# B&R Automation Studio project TD52 (part 122)

### module_HC.typ - Package data types
```iecst
TYPE
	IN_HC_Struct : 	STRUCT
		tAB2HC : AmmBase2MM;
		tPB2MM : ParaBase2MM_type;
		tCtr_Cust1_Out : _tGeACtrOut; (*controller customized*) (*OldName:REG1; Cycle:5;*)
		tCtr_Cust2_Out : _tGeACtrOut; (*controller customized*) (*OldName:REG2; Cycle:5;*)
		tCtr_Cust3_Out : _tGeACtrOut; (*controller customized*) (*OldName:REG3; Cycle:5;*)
		tCtr_Cust4_Out : _tGeACtrOut; (*controller customized*) (*OldName:REG4; Cycle:5;*)
		tCtr_Cust5_Out : _tGeACtrOut; (*controller customized*) (*OldName:REG5; Cycle:5;*)
		tCtr_Cust6_Out : _tGeACtrOut; (*controller customized*) (*OldName:REG6; Cycle:5;*)
		tCtr_Cust7_Out : _tGeACtrOut; (*controller customized*) (*OldName:REG7; Cycle:5;*)
		tCtr_Cust8_Out : _tGeACtrOut; (*controller customized*) (*OldName:REG8; Cycle:5;*)
		tCtr_Cust1_In : _tGeACtrIn; (*controller customized*) (*OldName:F_SPSR1; Cycle:5;*)
		tCtr_Cust2_In : _tGeACtrIn; (*controller customized*) (*OldName:F_SPSR2; Cycle:5;*)
		tCtr_Cust3_In : _tGeACtrIn; (*controller customized*) (*OldName:F_SPSR3; Cycle:5;*)
		tCtr_Cust4_In : _tGeACtrIn; (*controller customized*) (*OldName:F_SPSR4; Cycle:5;*)
		tCtr_Cust5_In : _tGeACtrIn; (*controller customized*) (*OldName:F_SPSR5; Cycle:5;*)
		tCtr_Cust6_In : _tGeACtrIn; (*controller customized*) (*OldName:F_SPSR6; Cycle:5;*)
		tCtr_Cust7_In : _tGeACtrIn; (*controller customized*) (*OldName:F_SPSR7; Cycle:5;*)
		tCtr_Cust8_In : _tGeACtrIn; (*controller customized*) (*OldName:F_SPSR8; Cycle:5;*)
		rCust_SparePara : ARRAY[0..200]OF REAL; (*SPS_REZP1 to SPS_REZP200	*) (* OldName: SPS_REZP1, SPS_REZP2, SPS_REZP70; Cycle: 5; *)
		tCustAnaIn : ARRAY[0..120]OF HALioAi_Type; (*Replacement for RAN_KANAL...*) (*OldName: ANA_RAN	; Cycle: 5;*)
		tCustDigIn : ARRAY[0..200]OF HALioDi_Type; (*new, reserved for Project specific use*) (*OldName: new PV	; Cycle: 5;*)
		tT_ECW_Ext_Hi : HALioDi_Type; (*DI temperature engine cooling water high external*) (*OldName:KTMA; Cycle:5;*)
		tEC_Failure : HALioDi_Type; (*DI emergency cooler failure*) (*OldName:ST_K; Cycle:5;*)
		tChC_Failure : HALioDi_Type; (*DI charge cooler failure*) (*OldName:ST_GKV; Cycle:5;*)
		tPr_CCircuit_Lo : HALioDi_Type; (*DI water pressure cooler circuit low*) (*OldName:WDK; Cycle:5;*)
		tPr_HW_Lo : HALioDi_Type; (*DI heat water pressure low*) (*OldName:HWD; Cycle:5;*)
		tPr_ChC_Lo : HALioDi_Type; (*DI charge cooler water pressure low*) (*OldName:GKWD; Cycle:5;*)
		tGCB_On : HALioDi_Type; (*DI generator circuit breaker closed*) (*OldName:GCB_ON; Cycle:5;*)
		tT_AirOutdoor : HALioAi_Type; (*AI temperature air outdoor*) (*OldName:ANA_ULT; Cycle:5;*)
		tPr_ECW : HALioAi_Type; (*pressure engine cooling water M.04-PI-001*) (*OldName:ANA.KWD; Cycle:5;*)
		tPr_ECWaEng : HALioAi_Type; (*pressure engine cooling water after engine M.04-PI-058*) (*OldName:AI_p_ECWaEng; Cycle:5;*)
		tT_ECW : HALioAi_Type; (*temperature engine cooling water M.04-TI-001*) (*OldName:ANA.KWT; Cycle:5;*)
		tT_HW_ReBeEng : HALioAi_Type; (*temperature heat water return before engine M.06-TI-001*) (*OldName:ANA.RLT_M; Cycle:5;*)
		tT_HW_ReAfEC : HALioAi_Type; (*temperature heat water return after emergency cooler P.06-TI-015, M.04-TI-015*) (*OldName:ANA.RLT_NK; Cycle:5;*)
		tT_HW_Re : HALioAi_Type; (*temperature heat water return P.06-TI-012, M.04-TI-012*) (*OldName:ANA.RLTP; Cycle:5;*)
		tT_HW_Su : HALioAi_Type; (*temperature heat water supply P.06-TI-014, M.04-TI-014*) (*OldName:ANA.VLTP; Cycle:5;*)
		tT_Su_PriCirc : HALioAi_Type; (*AI supply water temperature primary circuit [°C]*) (*OldName: new PV	; Cycle: 5;*)
		tT_Re_PriCirc : HALioAi_Type; (*AI return water temperature primary circuit [°C]*) (*OldName: new PV	; Cycle: 5;*)
		tT_Su_SecCirc : HALioAi_Type; (*AI supply water temperature secondary circuit [°C]*) (*OldName: new PV	; Cycle: 5;*)
		tT_Re_SecCirc : HALioAi_Type; (*AI return water temperature secondary circuit [°C]*) (*OldName: new PV	; Cycle: 5;*)
		tP_Heat : HALioAi_Type; (*AI heating power engine heat water circuit [kW]*) (*OldName: new PV	; Cycle: 5;*)
		tP_Heat_Imp : HALioDi_Type; (*DI heating power engine heat water circuit pulse*) (*OldName: new PV	; Cycle: 5;*)
		rT_Ch_T2s_Avg : REAL; (*average charge temperature t2' [°C]*) (*OldName: newPV; Cycle: 5;*)
		tT_EO : HALioAi_Type; (*temperature engine oil M.03-TI-001*) (*OldName:ANA.OTP; Cycle:5;*)
		tECWP1Dem : HALioDo_Type; (*DO engine cooling water pump 1 demand*) (*OldName:A_MKWP1; Cycle:5;*)
		tPr_HW_Hi1 : HALioDi_Type; (*DI heat water pressure high*) (*OldName:HWDX1; Cycle:5;*)
		tPr_HW_Hi : HALioDi_Type; (*DI heat water pressure high*) (*OldName:HWDX; Cycle:5;*)
		tT_HW_Hi1 : HALioDi_Type; (*DI heat water temperature high P.06-TS-023*) (*OldName:HWTP1; Cycle:5;*)
		tT_HW_Hi : HALioDi_Type; (*DI heat water temperature high P.06-TS-001*) (*OldName:HWTP; Cycle:5;*)
		tFlow_HW_Lo : HALioDi_Type; (*DI heat water flow low*) (*OldName:HWDF; Cycle:5;*)
		tT_ChCW_Hi : HALioDi_Type; (*DI charge cooling water temperature high*) (*OldName:GKWT_2; Cycle:5;*)
		tT_HW_Su_LT : HALioAi_Type; (*temperature heat water supply low temp.circuit [°C] M.07-TI-048*) (*OldName:NT_supply_water_temp; Cycle:5;*)
		tT_ECW_AfEng : HALioAi_Type; (*temperature engine cooling water after engine [°C]*) (*OldName:MKW_press_after_engine; Cycle:5;*)
		tEng_Run : HALioDo_Type; (*engine is running*) (*OldName:M_BTRB; Cycle:5;*)
		tT_HW_Re_LT : HALioAi_Type; (*temperature heat water return low temp.circuit [°C] M.07-TI-001*) (*OldName:iT_HWR_LT; Cycle:5;*)
		tAuxV_ModIf_ok : HALioDi_Type; (*DI auxiliary voltage supply ok Module interface*) (*OldName:SPG_HBT; Cycle:5;*)
		tAuxV_Aux_ok : HALioDi_Type; (*DI auxiliary voltage supply ok Auxiliaries panel*) (*OldName:SPG_HBT; Cycle:5;*)
		tAuxV_Supply_Ok : HALioDi_Type; (*DI auxiliary voltage supply ok*) (*OldName:SPG_HBT; Cycle:5;*)
		tChC_FanRdy : HALioDi_Type; (*DI charge cooler fan ready*) (*OldName:RDY_ICF; Cycle:5;*)
		tPr_HW_Su_LT : HALioAi_Type; (*supply water pressure LT circuit M.07-PI-001*) (*OldName:AI_p_VL_NT; Cycle:5;*)
		tPr_HW_Su_HT : HALioAi_Type; (*supply water pressure HT circuit M.06-PI-001*) (*OldName:AI_p_VL_HT; Cycle:5;*)
		tT_ECWbEng : HALioAi_Type; (*engine cooling water temperature before engine measurement active M.04-TI-002*) (*OldName:newPv; Cycle:5;*)
		tPr_HW_Re_LT : HALioAi_Type; (*pressure heat water return low temp.circuit M.07-PI-002*) (*OldName:newPv; Cycle:5;*)
		tPr_HW_Re_HT : HALioAi_Type; (*pressure heat water return high temp.circuit M.06-PI-002*) (*OldName:newPv; Cycle:5;*)
		tPr_HW_Re_PreH_ECW : HALioAi_Type; (*pressure heat water return preheating engine cooling water M.04-PI-005*) (*OldName:newPv; Cycle:5;*)
		tPr_HW_Re_PreH_EO : HALioAi_Type; (*pressure heat water return preheating engine oil M.03-PI-005*) (*OldName:newPv; Cycle:5;*)
		tPr_EO_Mod_Out : HALioAi_Type; (*pressure engine oil module outlet M.03-PI-006*) (*OldName:newPv; Cycle:5;*)
		tT_ECW_Mod_In : HALioAi_Type; (*temperature engine cooling water, engine cooling water module inlet M.04-TI-003*) (*OldName:newPv; Cycle:5;*)
		tT_ECW_Mod_Out : HALioAi_Type; (*temperature engine cooling water, engine cooling water module outlet M.04-TI-004*) (*OldName:newPv; Cycle:5;*)
		tT_EO_Mod_In : HALioAi_Type; (*temperature engine oil, oil module inlet M.03-TI-004*) (*OldName:newPv; Cycle:5;*)
		tT_EO_Mod_Out : HALioAi_Type; (*temperature engine oil, oil module outlet M.03-TI-003*) (*OldName:newPv; Cycle:5;*)
		tT_HW_Su_PreH_ECW : HALioAi_Type; (*temperature heat water supply preheating engine cooling water M.04-TI-005*) (*OldName:newPv; Cycle:5;*)
		tT_HW_Re_PreH_ECW : HALioAi_Type; (*temperature heat water return preheating engine cooling water M.04-TI-006*) (*OldName:newPv; Cycle:5;*)
		tT_HW_Su_PreH_EO : HALioAi_Type; (*temperature heat water supply preheating engine oil M.03-TI-005*) (*OldName:newPv; Cycle:5;*)
		tT_HW_Re_PreH_EO : HALioAi_Type; (*temperature heat water return preheating engine oil M.03-TI-006*) (*OldName:newPv; Cycle:5;*)
		iSt_OpMode : UDINT; (*engine operating mode*) (*OldName:newPv; Cycle:5;*)
		rN_EngAct : REAL; (*engine speed actual [1/min]*) (*OldName:n_ist; Cycle:5;*)
		rT_ChC_Ctr_Wex : REAL; (*charge temperature controller external setpoint(knocking)*) (*OldName:Wex_GEMREG; Cycle:5;*)
		bEng_Dem_EPS : BOOL; (*engine demand for emergency power supply*) (*OldName:M_NANF; Cycle:5;*)
		bEng_Aux_Dem_CDR : BOOL; (*engine auxiliaries demand with cool down run*) (*OldName:ANFHBT; Cycle:5;*)
		bEng_Aux_Dem : BOOL; (*engine auxiliaries demand*) (*OldName:M_ANFHBT; Cycle:5;*)
		iIdx_OMSS : INT; (*engine operation mode selection*) (*OldName:newPv; Cycle:5;*)
		rP_Act_Norm_Filt : REAL; (*actual power related to rP_Nom filtered(1s) [%] *) (*OldName:P_IST; Cycle:5;*)
		bEC_Rel : BOOL; (*release emergency cooler from monitoring*) (*OldName:K_frg; Cycle:5;*)
		bChC_Rel : BOOL; (*release charge cooler from monitoring*) (*OldName:GK_frg; Cycle:5;*)
		tCDP_Dem : HALioDo_Type; (*demand condensor pump*) (*OldName:newPv; Cycle:5;*)
		tHWF_Fail : HALioDi_Type; (*failure heating circuit flap*) (*OldName:newPv; Cycle:5;*)
		tCDP_Op : HALioDi_Type; (*failure condensor pump*) (*OldName:newPv; Cycle:5;*)
		tT_HW_HC_Re : HALioAi_Type; (*heating circuit return temperature*) (*OldName:newPv; Cycle:5;*)
		tT_CD_Su : HALioAi_Type; (*supply temperature condensor circuit*) (*OldName:newPv; Cycle:5;*)
		tT_CD_Re : HALioAi_Type; (*return temperature condensor circuit*) (*OldName:newPv; Cycle:5;*)
		tPos_HW_ReValve : HALioAi_Type; (*position heating water return temperature regulation valve*) (*OldName:newPv; Cycle:5;*)
		tPos_HW_EC_ReValve : HALioAi_Type; (*position heating water return temperature after cooler regulation valve*) (*OldName:newPv; Cycle:5;*)
		tPos_ChC_Valve : HALioAi_Type; (*position charge temperature regulation valve*) (*OldName:newPv; Cycle:5;*)
		tBHV_Op : HALioDi_Type; (*failure boiler house ventilation*) (*OldName:newPv; Cycle:5;*)
		tDemnd_BHV : HALioDi_Type; (*demand boiler house ventilation*) (*OldName:newPv; Cycle:5;*)
		bMsg1031 : BOOL; (*emergency stop / safety loop*) (*OldName:M_SIS; Cycle:5;*)
		bMsg1053 : BOOL; (*gas alarm*) (*OldName:M_GAL; Cycle:5;*)
		bMsg1054 : BOOL; (*fire alarm*) (*OldName:M_BAL; Cycle:5;*)
		bMsg3003 : BOOL; (*signal failure( 2101 or 2102 or 2103 or 2104 or 3152 > 24h)*) (*OldName:M_MS; Cycle:5;*)
		tManAuxCtr : tManAuxCtr_typ; (*Manual operating auxiliaries control - Handbedienebene*) (*OldName: new PV; Cycle: 5;*)
		tT_ECW_bChC_HT : HALioAi_Type; (*temperature engine cooling water before charge cooler high temp.circ. M.06-TI-014*) (*OldName:newPv; Cycle:5;*)
		tT_ECW_bOilC : HALioAi_Type; (*temperature engine cooling water before oil cooler M.06-TI-020*) (*OldName:newPv; Cycle:5;*)
		tT_ECW_bECWC : HALioAi_Type; (*temperature engine cooling water before engine cooling water cooler M.06-TI-030*) (*OldName:newPv; Cycle:5;*)
		bAMM_T_Ch_T2s_Avg : BOOL; (*collective warning - average charge temp. t2'  *) (*OldName: new PV; Cycle:5;*) (*SWAT920/2*)
		bT_ChC_Ctr_Wex_Enable_Cust : BOOL; (*new V4.5*)
		rT_ChC_Ctr_Wex_Cust : REAL; (*new V4..5*)
		rCustomizedHC : ARRAY[0..99]OF REAL; (*New customizable interface 2017  - BETA PHASE, use only in coordination with TPSS*)
		bChC2_Rel : BOOL; (*release charge cooler 2 from monitoring*) (*OldName:newPV; Cycle:5;*)
		bAMM_T_Ch_T1HP_Avg : BOOL; (*collective warning - average charge temp. before high-pressure TC*) (*OldName: new PV; Cycle:5;*)
		rT_Ch_T1HP_Avg : REAL; (*average charge temperature before high-pressure turbo charger T1-HP [°C]*) (*OldName: newPV; Cycle: 5;*)
		tPos_ChC2_Valve : HALioAi_Type; (*AI Position temperature-regulation-valve 2nd LT charge cooler circuit (T1-HP)*) (*OldName:newPv; Cycle:5;*)
		tPr_ChC2_Lo : HALioDi_Type; (*DI charge cooler 2 water pressure low - DI = FALSE if pressure is low*) (*OldName:newPV; Cycle:5;*)
		tChC2_FanRdy : HALioDi_Type; (*DI charge cooler 2 fan ready*) (*OldName:newPV; Cycle:5;*)
		tChC2_Failure : HALioDi_Type; (*DI charge cooler 2 failure - DI = FALSE if failure active*) (*OldName:newPV; Cycle:5;*)
		tT_ChC2_Su_LT : HALioAi_Type; (*AI supply water temperature 2nd LT charge cooler circuit (T1-HP) [°C] (P.07-TI-004)*) (*OldName:newPV; Cycle:5;*)
		tT_ChC2_Re_LT : HALioAi_Type; (*AI return water temperature 2nd LT charge cooler circuit (T1-HP) [°C] (P.07-TI-006)*) (*OldName:newPV; Cycle:5;*)
		tT_ChC2W_Hi : HALioDi_Type; (*DI charge cooler 2 water temperature high - DI = FALSE if water temp. too high*) (*OldName:newPV; Cycle:5;*)
		tT_HW_EGHE_Hi : HALioDi_Type; (*DI Heating water temperature max. exhaust gas cooler*)
		tT_HW_EGCD_Hi : HALioDi_Type; (*DI Heating water temperature max. exhaust gas condenser*)
		tCust_HW_Ext_Trip : HALioDi_Type; (*DI External heating water circuit monitoring*)
		bECWP_MechDriven : BOOL;  (* CUSTOM for new Pr_ECW plausibility check: Mechanically driven ECWP on type3 or type2 *)
		tECWP_Op : HALioDi_Type; (* DI engine cooling water pump operating *)
		tT_HW_Su_Unit : HALioAi_Type; (*SAFETY PLC: Heating water supply temperature - Unit (M.06-TI-003)*) (*OldName: new PV; Cycle: 5;*) (*V04.25.00.00*)
	END_STRUCT; (*END_IN*)
	OUT_HC_Struct : 	STRUCT
		tChC_Heating : HALioDo_Type; (*DO charge cooler pre heating*) (*OldName:FG_KT; Cycle:5;*)
		tHC2AB : MM2AmmBase;
		tHC2PB : MM2ParaBase_type;
		tExCo_Rel : HALioDo_Type; (*DO external cooler release*) (*OldName:FG_KT; Cycle:5;*)
		tChC_DemPump : HALioDo_Type; (*DO charge cooler demand pump*) (*OldName:GKP_EIN; Cycle:5;*)
		tChC_DemFan1 : HALioDo_Type; (*DO charge cooler demand fan 1*) (*OldName:GKV_1; Cycle:5;*)
		tChC_DemFan2 : HALioDo_Type; (*DO charge cooler demand fan 2*) (*OldName:GKV_2; Cycle:5;*)
		tChC_DemFan3 : HALioDo_Type; (*DO charge cooler demand fan 3*) (*OldName:GKV_3; Cycle:5;*)
		tChC_DemFan4 : HALioDo_Type; (*DO charge cooler demand fan 4*) (*OldName:GKV_4; Cycle:5;*)
		tChC_DemFan5 : HALioDo_Type; (*DO charge cooler demand fan 5*) (*OldName:GKV_5; Cycle:5;*)
		tChC_DemFan6 : HALioDo_Type; (*DO charge cooler demand fan 6*) (*OldName:GKV_6; Cycle:5;*)
		tChC_DemFan7 : HALioDo_Type; (*DO charge cooler demand fan 7*) (*OldName:GKV_7; Cycle:5;*)
		tChC_DemFan8 : HALioDo_Type; (*DO charge cooler demand fan 8*) (*OldName:GKV_8; Cycle:5;*)
		tChC_DemFan9 : HALioDo_Type; (*DO charge cooler demand fan 9*) (*OldName:GKV_9; Cycle:5;*)
		tChC_DemFan10 : HALioDo_Type; (*DO charge cooler demand fan 10*) (*OldName:GKV_10; Cycle:5;*)
		tChC_DemFan11 : HALioDo_Type; (*DO charge cooler demand fan 11*) (*OldName:GKV_11; Cycle:5;*)
		tChC_DemFan12 : HALioDo_Type; (*DO charge cooler demand fan 12*) (*OldName:GKV_12; Cycle:5;*)
		tChC_DemFan13 : HALioDo_Type; (*DO charge cooler demand fan 13*) (*OldName:GKV_13; Cycle:5;*)
		tChC_DemFan14 : HALioDo_Type; (*DO charge cooler demand fan 14*) (*OldName:GKV_14; Cycle:5;*)
		tChC_DemFan15 : HALioDo_Type; (*DO charge cooler demand fan 15*) (*OldName:GKV_15; Cycle:5;*)
		tChC_DemFan16 : HALioDo_Type; (*DO charge cooler demand fan 16*) (*OldName:GKV_16; Cycle:5;*)
		tEC_DemPump : HALioDo_Type; (*DO emergency cooler demand pump*) (*OldName:KP_EIN; Cycle:5;*)
		tEC_DemFan1 : HALioDo_Type; (*DO emergency cooler demand fan 1*) (*OldName:KV_1; Cycle:5;*)
		tEC_DemFan2 : HALioDo_Type; (*DO emergency cooler demand fan 2*) (*OldName:KV_2; Cycle:5;*)
		tEC_DemFan3 : HALioDo_Type; (*DO emergency cooler demand fan 3*) (*OldName:KV_3; Cycle:5;*)
		tEC_DemFan4 : HALioDo_Type; (*DO emergency cooler demand fan 4*) (*OldName:KV_4; Cycle:5;*)
		tEC_DemFan5 : HALioDo_Type; (*DO emergency cooler demand fan 5*) (*OldName:KV_5; Cycle:5;*)
		tEC_DemFan6 : HALioDo_Type; (*DO emergency cooler demand fan 6*) (*OldName:KV_6; Cycle:5;*)
		tEC_DemFan7 : HALioDo_Type; (*DO emergency cooler demand fan 7*) (*OldName:KV_7; Cycle:5;*)
		tEC_DemFan8 : HALioDo_Type; (*DO emergency cooler demand fan 8*) (*OldName:KV_8; Cycle:5;*)
		tEC_DemFan9 : HALioDo_Type; (*DO emergency cooler demand fan 9*) (*OldName:KV_9; Cycle:5;*)
		tEC_DemFan10 : HALioDo_Type; (*DO emergency cooler demand fan 10*) (*OldName:KV_10; Cycle:5;*)
		tEC_DemFan11 : HALioDo_Type; (*DO emergency cooler demand fan 11*) (*OldName:KV_11; Cycle:5;*)
		tEC_DemFan12 : HALioDo_Type; (*DO emergency cooler demand fan 12*) (*OldName:KV_12; Cycle:5;*)
		tEC_DemFan13 : HALioDo_Type; (*DO emergency cooler demand fan 13*) (*OldName:KV_13; Cycle:5;*)
		tEC_DemFan14 : HALioDo_Type; (*DO emergency cooler demand fan 14*) (*OldName:KV_14; Cycle:5;*)
		tEC_DemFan15 : HALioDo_Type; (*DO emergency cooler demand fan 15*) (*OldName:KV_15; Cycle:5;*)
		tEC_DemFan16 : HALioDo_Type; (*DO emergency cooler demand fan 16*) (*OldName:KV_16; Cycle:5;*)
		tECW_DemBpP : HALioDo_Type; (*DO demand engine cooling water bypass pump (AMOT)*) (*OldName:BP_P; Cycle:5;*)
		tECW_DemBpV : HALioDo_Type; (*DO demand engine cooling water bypass valve (AMOT)*) (*OldName:BP_V; Cycle:5;*)
		tCtr_ChC_Set : HALioAo_Type; (*AO charge temperature cooler control valve*) (*OldName:Reg9_y; Cycle:5;*)
		tCtr_HWRe_Set : HALioAo_Type; (*AO heat water return temperature control valve*) (*OldName:Reg10_y; Cycle:5;*)
		tCtr_EC_Set : HALioAo_Type; (*AO heat water return temperature control valve emergency cooler*) (*OldName:Reg11_y; Cycle:5;*)
		tCtr_HWSu_Set : HALioAo_Type; (*AO heat water supply temperature control valve*) (*OldName:Reg14_y; Cycle:5;*)
		tCtr_ChCV_Set : HALioAo_Type; (*AO charge temperature cooler ventilation*) (*OldName:Reg15_y, GKV_y; Cycle:5;*)
		tCtr_ChCHP_Set : HALioAo_Type; (*AO charge temperature cooler high pressure control valve*) (*OldName:Reg18_y; Cycle:5;*)
		bT_ECW_Hi : BOOL; (*temperature engine cooling water limit high*) (*OldName:AN_KTMA; Cycle:5;*)
		bT_ECW_Lo : BOOL; (*temperature engine cooling water limit low*) (*OldName:AN_KTMI; Cycle:5;*)
		bT_ECW_RelLoad : BOOL; (*temperature engine cooling water release load*) (*OldName:AN_LFG; Cycle:5;*)
		bT_ECW_PreH_OFF : BOOL; (*temperature engine cooling water preheating off*) (*OldName:AN_VORW; Cycle:5;*)
		rP_Red_T_HWR_Norm : REAL; (*power reduction heat water return temperature high [% Pnom]*) (*OldName:RED_RLT; Cycle:5;*)
		rP_Red_T_ECW_Norm : REAL; (*power reduction engine cooling water temperature high [% Pnom]*) (*OldName:RED_KWT; Cycle:5;*)
		bPr_ECW_Lo1 : BOOL; (*pressure engine cooling water limit low 1*) (*OldName:AN_KDGW1; Cycle:5;*)
		tHWF_Dem : HALioDo_Type; (*demand heating circuit flap*) (*OldName:newPv; Cycle:5;*)
		tCtr_CDSu_Set : HALioAo_Type; (*setpoint frequency conferter condensor pump*) (*OldName:newPv; Cycle:5;*)
		tBHV_Dem : HALioDo_Type; (*demand boiler house ventilation*) (*OldName:newPv; Cycle:5;*)
		iCnt_P_Heat : DINT; (*counter heating power engine heat water circuit*) (*OldName:newPv; Cycle:5;*)
		bMsg1019 : BOOL; (*engine cooling water pressure low*) (*OldName:M_KDMI; Cycle:5;*)
		bMsg2104 : BOOL; (*signal failure engine cooling water pressure *) (*OldName:M_MSKWD; Cycle:5;*)
		bMsg2101 : BOOL; (*signal failure engine cooling water temperature*) (*OldName:M_MSKWT; Cycle:5;*)
		bMsg3404 : BOOL; (*water pressure cooler circuit low*) (*OldName:M_NKWD_W; Cycle:5;*)
		bMsg1130 : BOOL; (*charge cooler water pressure low*) (*OldName:AMM_A11xx[]; Cycle:5;*)
		bMsg2117 : BOOL; (*charge cooler water pressure low*) (*OldName:M_GKWD; Cycle:5;*)
		rP_Red_T_ECW_Low_Norm : REAL; (*power reduction engine cooling water temperature low [% Pnom]*) (*OldName:newPv; Cycle:5;*)
		rCustomizedHC : ARRAY[0..99]OF REAL; (*New customizable interface 2017  - BETA PHASE, use only in coordination with TPSS*)
		tChC2_DemPump : HALioDo_Type; (*DO charge cooler 2 demand pump*) (*OldName:newPV; Cycle:5;*)
		tCtr_ChC2_Valve_Set : HALioAo_Type; (*AO Control temperature-regulation-valve 2nd LT charge cooler circuit (T1-HP)*) (*OldName:newPV; Cycle:5;*)
		tChC2_DemFan1 : HALioDo_Type; (*DO charge cooler 2 demand fan 1*) (*OldName:newPV; Cycle:5;*)
		tChC2_DemFan2 : HALioDo_Type; (*DO charge cooler 2 demand fan 2*) (*OldName:newPV; Cycle:5;*)
		tChC2_DemFan3 : HALioDo_Type; (*DO charge cooler 2 demand fan 3*) (*OldName:newPV; Cycle:5;*)
		tChC2_DemFan4 : HALioDo_Type; (*DO charge cooler 2 demand fan 4*) (*OldName:newPV; Cycle:5;*)
		tChC2_DemFan5 : HALioDo_Type; (*DO charge cooler 2 demand fan 5*) (*OldName:newPV; Cycle:5;*)
		tChC2_DemFan6 : HALioDo_Type; (*DO charge cooler 2 demand fan 6*) (*OldName:newPV; Cycle:5;*)
		tChC2_DemFan7 : HALioDo_Type; (*DO charge cooler 2 demand fan 7*) (*OldName:newPV; Cycle:5;*)
		tChC2_DemFan8 : HALioDo_Type; (*DO charge cooler 2 demand fan 8*) (*OldName:newPV; Cycle:5;*)
		tChC2_DemFan9 : HALioDo_Type; (*DO charge cooler 2 demand fan 9*) (*OldName:newPV; Cycle:5;*)
		tChC2_DemFan10 : HALioDo_Type; (*DO charge cooler 2 demand fan 10*) (*OldName:newPV; Cycle:5;*)
		tChC2_DemFan11 : HALioDo_Type; (*DO charge cooler 2 demand fan 11*) (*OldName:newPV; Cycle:5;*)
		tChC2_DemFan12 : HALioDo_Type; (*DO charge cooler 2 demand fan 12*) (*OldName:newPV; Cycle:5;*)
		tChC2_DemFan13 : HALioDo_Type; (*DO charge cooler 2 demand fan 13*) (*OldName:newPV; Cycle:5;*)
		tChC2_DemFan14 : HALioDo_Type; (*DO charge cooler 2 demand fan 14*) (*OldName:newPV; Cycle:5;*)
		tChC2_DemFan15 : HALioDo_Type; (*DO charge cooler 2 demand fan 15*) (*OldName:newPV; Cycle:5;*)
		tChC2_DemFan16 : HALioDo_Type; (*DO charge cooler 2 demand fan 16*) (*OldName:newPV; Cycle:5;*)
		bMsg9226 : BOOL; (*charge cooler 2 water pressure low*) (*OldName:newPV; Cycle:5;*)
		tChC2_Heating : HALioDo_Type; (*DO Demand charge cooler 2 pre heating*) (*OldName:newPV; Cycle:5;*)
		bMsg2684 : BOOL; (*Temperature heat water supply hydraulic engine cooling water preheating signal failure*) (*OldName:newPV; Cycle:5;*)
		bCCWP_Dem : BOOL; (*Charge cooler water pump demand*) (*OldName:newPV; Cycle:5;*)
		bCC2WP_Dem : BOOL; (*Charge cooler 2 water pump demand*) (*OldName:newPV; Cycle:5;*)
		bEmCWP_Dem : BOOL; (*Emergency cooler water pump demand*) (*OldName:newPV; Cycle:5;*)
		bMsg1050 : BOOL; (*engine cooling water pressure high*) (*OldName:newPV; Cycle:5;*)
		tECW_ShutOffVal_Dem : HALioDo_Type; (*demand 2-way shut off valve engine jacket water circuit*)
		tValHeater_Dem : HALioDo_Type; (*demand 3-way valve heater*)
		tFanRingHeater_Dem : HALioDo_Type; (*demand fan ring heater*)
	END_STRUCT; (*END_OUT*)
	VIS2MM_Struct : 	STRUCT
		tCtr_CDSu_In : _tGeACtrIn; (*condensor circuit supply temperature controller*) (*OldName:newPv; Cycle:5;*)
		tCtr_ChC_In : _tGeACtrIn; (*charge temperature controller*) (*OldName:REG9; Cycle:5;*)
		tCtr_HWRe_In : _tGeACtrIn; (*heat water return temperature controller*) (*OldName:REG10; Cycle:5;*)
		tCtr_EC_In : _tGeACtrIn; (*emergency cooler controller*) (*OldName:REG11; Cycle:5;*)
		tCtr_HWSu_In : _tGeACtrIn; (*heat water supply temperature controller*) (*OldName:REG14; Cycle:5;*)
		tCtr_ChCV_In : _tGeACtrIn; (*charge cooler ventilation controller*) (*OldName:REG15; Cycle:5;*)
		tCtr_ChCHP_In : _tGeACtrIn; (*charge temperature high pressure controller*) (*OldName:REG18; Cycle:5;*)
		tCtr_ChC_T1HP_In : _tGeACtrIn; (*charge temperature before high-pressure turbo charger controller*) (*OldName:newPV; Cycle:5;*)
	END_STRUCT; (*END_VIS2MM*)
	MM2VIS_Struct : 	STRUCT
		tCtr_CDSu_Out : _tGeACtrOut; (*condensor circuit supply temperature controller*) (*OldName:newPv; Cycle:5;*)
		tCtr_ChC_Out : _tGeACtrOut; (*charge temperature controller*) (*OldName:REG9; Cycle:5;*)
		tCtr_HWRe_Out : _tGeACtrOut; (*heat water return temperature controller*) (*OldName:REG10; Cycle:5;*)
		tCtr_EC_Out : _tGeACtrOut; (*emergency cooler controller*) (*OldName:REG11; Cycle:5;*)
		tCtr_HWSu_Out : _tGeACtrOut; (*heat water supply temperature controller*) (*OldName:REG14; Cycle:5;*)
		tCtr_ChCV_Out : _tGeACtrOut; (*charge cooler ventilation controller*) (*OldName:REG15; Cycle:5;*)
		tCtr_ChCHP_Out : _tGeACtrOut; (*charge temperature high pressure controller*) (*OldName:REG18; Cycle:5;*)
		rT_AirOutdoor : REAL; (*temperature air outdoor *) (*OldName:ANA_ULT; Cycle:5;*)
		bECW_DemBpP : BOOL; (*demand engine cooling water bypass pump*) (*OldName:BP_P; Cycle:5;*)
		bEC_Stage1 : BOOL; (*emergency cooler stage 1*) (*OldName:B_SV[38]; Cycle:5;*)
		bEC_Stage2 : BOOL; (*emergency cooler stage 2*) (*OldName:B_SV[39]; Cycle:5;*)
		bEC_Dem : BOOL; (*emergency cooler demanded*) (*OldName:newPv; Cycle:5;*)
		iSumChC_Stages : INT; (*summary charge cooler stages*) (*OldName:AnzGkuehlSt; Cycle:5;*)
		iSumEC_Stages : INT; (*summary emergency cooler stages*) (*OldName:AnzKuehlSt; Cycle:5;*)
		iCnt_P_Heat : DINT; (*counter heating power engine heat water circuit*) (*OldName:newPv; Cycle:5;*)
		rT_HW_ReBeEng : REAL; (*temperature heat water return before engine [°C]*) (*OldName:ANA.RLT_M; Cycle:5;*)
		rT_HW_ReAfEC : REAL; (*temperature heat water return after emergency cooler [°C]*) (*OldName:ANA.RLT_NK; Cycle:5;*)
		rT_HW_Re : REAL; (*temperature heat water return [°C]*) (*OldName:ANA.RLTP; Cycle:5;*)
		rT_HW_Su : REAL; (*temperature heat water supply [°C]*) (*OldName:ANA.VLTP; Cycle:5;*)
		rPr_HW_Su_HT : REAL; (*pressure heat water supply high temp.circuit [bar]*) (*OldName:AI_p_VL_HT; Cycle:5;*)
		rPr_ECW : REAL; (*pressure engine cooling water [°C]*) (*OldName:ANA.KWD; Cycle:5;*)
		rPr_ECWaEng : REAL; (*pressure engine cooling water after engine [°C]*) (*OldName:MKWPress_a_e; Cycle:5;*)
		rT_ECW : REAL; (*temperature engine cooling water [°C]*) (*OldName:ANA.KWT; Cycle:5;*)
		rP_Red_T_HWR_Norm : REAL; (*power reduction heat water return temperature high [% Pnom]*) (*OldName:ssPowerRedRLT; Cycle:5;*)
		rP_Red_T_ECW_Norm : REAL; (*power reduction engine cooling water temperature high [% Pnom]*) (*OldName:ssPowerRedKWT; Cycle:5;*)
		rT_HW_Su_LT : REAL; (*temperature heat water supply low temp.circuit [°C]*) (*OldName:NTemp_supply; Cycle:5;*)
		rPr_HW_Su_LT : REAL; (*pressure heat water supply low temp.circuit [bar]*) (*OldName:AI_p_VL_NT; Cycle:5;*)
		rT_ECW_AfEng : REAL; (*temperature engine cooling water after engine [°C]*) (*OldName:MKW_press_after_engine; Cycle:5;*)
		rT_HW_Re_LT : REAL; (*temperature heat water return low temp.circuit [°C]*) (*OldName:iT_HWR_LT; Cycle:5;*)
		rT_ECWbEng : REAL; (*engine cooling water temperature before engine M.04-TI-002*) (*OldName:newPv; Cycle:5;*)
		rPr_HW_Re_LT : REAL; (*pressure heat water return low temp.circuit M.07-PI-002*) (*OldName:newPv; Cycle:5;*)
		rPr_HW_Re_HT : REAL; (*pressure heat water return high temp.circuit M.06-PI-002*) (*OldName:newPv; Cycle:5;*)
		rPr_HW_Re_PreH_ECW : REAL; (*pressure heat water return preheating engine cooling water M.04-PI-005*) (*OldName:newPv; Cycle:5;*)
		rPr_HW_Re_PreH_EO : REAL; (*pressure heat water return preheating engine oil M.03-PI-005*) (*OldName:newPv; Cycle:5;*)
		rPr_EO_Mod_Out : REAL; (*pressure engine oil module outlet M.03-PI-006*) (*OldName:newPv; Cycle:5;*)
		rT_ECW_Mod_In : REAL; (*temperature  engine cooling water, engine cooling water module inlet M.04-TI-003*) (*OldName:newPv; Cycle:5;*)
		rT_ECW_Mod_Out : REAL; (*temperature  engine cooling water, engine cooling water module outlet M.04-TI-004*) (*OldName:newPv; Cycle:5;*)
		rT_EO_Mod_In : REAL; (*temperature engine oil, oil module inlet M.03-TI-004*) (*OldName:newPv; Cycle:5;*)
		rT_EO_Mod_Out : REAL; (*temperature engine oil, oil module outlet M.03-TI-003*) (*OldName:newPv; Cycle:5;*)
		rT_HW_Su_PreH_ECW : REAL; (*temperature heat water supply preheating engine cooling water M.04-TI-005*) (*OldName:newPv; Cycle:5;*)
		rT_HW_Re_PreH_ECW : REAL; (*temperature heat water return preheating engine cooling water M.04-TI-006*) (*OldName:newPv; Cycle:5;*)
		rT_HW_Su_PreH_EO : REAL; (*temperature heat water supply preheating engine oil M.03-TI-005*) (*OldName:newPv; Cycle:5;*)
		rT_HW_Re_PreH_EO : REAL; (*temperature heat water return preheating engine oil M.03-TI-006*) (*OldName:newPv; Cycle:5;*)
		rPos_HW_ReValve : REAL; (*position heating water return temperature regulation valve*) (*OldName:newPv; Cycle:5;*)
		rPos_HW_EC_ReValve : REAL; (*position heating water return temperature after cooler regulation valve*) (*OldName:newPv; Cycle:5;*)
		rPos_ChC_Valve : REAL; (*position charge temperature regulation valve*) (*OldName:newPv; Cycle:5;*)
		rT_Su_PriCirc : REAL; (*supply water temperature high primary circuit*) (*OldName:newPv; Cycle:5;*)
		rT_Re_PriCirc : REAL; (*return water temperature high primary circuit*) (*OldName:newPv; Cycle:5;*)
		rT_Su_SecCirc : REAL; (*supply water temperature high secondary circuit*) (*OldName:newPv; Cycle:5;*)
		rT_Re_SecCirc : REAL; (*return water temperature high secondary circuit*) (*OldName:newPv; Cycle:5;*)
		rP_Heat : REAL; (*heating power engine heat water circuit*) (*OldName:newPv; Cycle:5;*)
		bHWF_Dem : BOOL; (*demand heat circuit flap*) (*OldName:newPv; Cycle:5;*)
		rT_HW_HC_Re : REAL; (*heating circuit return temperature*) (*OldName:newPv; Cycle:5;*)
		bCDP_Dem : BOOL; (*demand condensor pump*) (*OldName:newPv; Cycle:5;*)
		bBHV_Dem : BOOL; (*demand boiler house ventilator*) (*OldName:newPv; Cycle:5;*)
		rT_CD_Re : REAL; (*return temperature condensor circuit [°C]*) (*OldName:newPv; Cycle:5;*)
		rT_CD_Su : REAL; (*supply temperature condensor circuit [°C]*) (*OldName:newPv; Cycle:5;*)
		bMsg1019 : BOOL; (*engine cooling water pressure low*) (*OldName:M_KDMI; Cycle:5;*)
		bMsg1021 : BOOL; (*engine cooling water temperature high*) (*OldName:M_KTMA; Cycle:5;*)
		bMsg1032 : BOOL; (*heat water  flow low*) (*OldName:M_HWDF; Cycle:5;*)
		bMsg1033 : BOOL; (*heat water  temperature high*) (*OldName:M_HWTP; Cycle:5;*)
		bMsg1034 : BOOL; (*heat water  pressure low*) (*OldName:M_HWD; Cycle:5;*)
		bMsg1035 : BOOL; (*heat water  pressure high*) (*OldName:M_HWDX; Cycle:5;*)
		bMsg1050 : BOOL; (*engine cooling water pressure high*) (*OldName:M_KDMA; Cycle:5;*)
		bMsg1063 : BOOL; (*heat water supply temperature high*) (*OldName:AMM_A10xx[]; Cycle:5;*)
		bMsg1070 : BOOL; (*signal failure heat water return temperature*) (*OldName:AMM_A10xx[]; Cycle:5;*)
		bMsg1071 : BOOL; (*signal failure heat water supply temperature*) (*OldName:AMM_A10xx[]; Cycle:5;*)
		bMsg1130 : BOOL; (*charge cooler water pressure low*) (*OldName:AMM_A11xx[]; Cycle:5;*)
		bMsg1145 : BOOL; (*engine cooling water temperature low*) (*OldName:AMM_W11xx[]; Cycle:5;*)
		bMsg1167 : BOOL; (*heat water return temperature high*) (*OldName:AMM_W11xx[]; Cycle:5;*)
		bMsg1186 : BOOL; (*signal failure heat water return temperature*) (*OldName:AMM_W11xx[]; Cycle:5;*)
		bMsg1187 : BOOL; (*signal failure heat water supply temperature*) (*OldName:AMM_W11xx[]; Cycle:5;*)
		bMsg2101 : BOOL; (*signal failure engine cooling water temperature*) (*OldName:AMM_W21xx[]; Cycle:5;*)
		bMsg2104 : BOOL; (*signal failure engine cooling water pressure*) (*OldName:AMM_W21xx[]; Cycle:5;*)
		bMsg2116 : BOOL; (*emergency cooler failure*) (*OldName:AMM_W21xx[]; Cycle:5;*)
		bMsg2117 : BOOL; (*charge cooler water pressure low*) (*OldName:M_GKWD; Cycle:5;*)
		bMsg2119 : BOOL; (*charge cooler failure*) (*OldName:AMM_W21xx[]; Cycle:5;*)
		bMsg2341 : BOOL; (*Heating water temperature maximum - exhaust gas cooler*) (*OldName:newPv; Cycle:5;*)
		bMsg2342 : BOOL; (*Heating water temperature maximum - exhaust gas condenser*) (*OldName:newPv; Cycle:5;*)
		bMsg2343 : BOOL; (*External heating water circuit monitoring tripped*) (*OldName:newPv; Cycle:5;*)
		bMsg2428 : BOOL; (*heat water  flow low*) (*SWAT920/1*)
		bMsg2429 : BOOL; (*heat water  temperature high*) (*SWAT920/1*)
		bMsg2430 : BOOL; (*heat water supply temperature high*) (*SWAT920/1*)
		bMsg2638 : BOOL; (*supply water pressure LT circuit signal failure*) (*OldName:AMM_W26xx[]; Cycle:5;*)
		bMsg2639 : BOOL; (*supply water pressure HT circuit signal failure*) (*OldName:AMM_W26xx[]; Cycle:5;*)
		bMsg2640 : BOOL; (*return water temperature LT circuit signal failure*) (*OldName:AMM_W26xx[]; Cycle:5;*)
		bMsg2641 : BOOL; (*supply water temperature LT circuit signal failure*) (*OldName:AMM_W26xx[]; Cycle:5;*)
		bMsg2647 : BOOL; (*engine  cooling water pressure after engine signal failure*) (*OldName:AMM_W26xx; Cycle:5*)
		bMsg2667 : BOOL; (*engine cooling water temperature before engine signal failure*) (*OldName:AMM_W26xx; Cycle:5*)
		bMsg2675 : BOOL; (*pressure heat water return low temperature circuit signal failure*)
		bMsg2676 : BOOL; (*pressure heat water return high temperature circuit signal failure*)
		bMsg2677 : BOOL; (*pressure heat water return hydraulic engine cooling water preheating signal failure*)
		bMsg2678 : BOOL; (*pressure heat water return hydraulic oil preheating signal failure*)
		bMsg2679 : BOOL; (*pressure oil module oil outlet signal failure*)
		bMsg2680 : BOOL; (*temperature engine cooling water module inlet  signal failure*)
		bMsg2681 : BOOL; (*temperature engine cooling water module outlet  signal failure*)
		bMsg2682 : BOOL; (*temperature oil module oil inlet signal failure*)
		bMsg2683 : BOOL; (*temperature oil module oil outlet  signal failure*)
		bMsg2684 : BOOL; (*temperature heat water supply hydraulic engine cooling water preheating signal failure*)
		bMsg2685 : BOOL; (*temperature heat water return hydraulic engine cooling water preheating signal failure*)
		bMsg2686 : BOOL; (*temperature heat water supply hydraulic oil preheating signal failure*)
		bMsg2687 : BOOL; (*temperature heat water return hydraulic oil preheating signal failure*)
		bMsg2710 : BOOL; (*measuring signal failure position control valve heat water return temperature*) (*OldName:newPv; Cycle:5;*)
		bMsg2711 : BOOL; (*measuring signal failure position control valve heat water return temperature after cooler*) (*OldName:newPv; Cycle:5;*)
		bMsg2712 : BOOL; (*measuring signal failure position control valve charge cooler circuit temperature*) (*OldName:newPv; Cycle:5;*)
		bMsg2713 : BOOL; (*measuring signal failure supply water temperature primary circuit*) (*OldName:newPv; Cycle:5;*)
		bMsg2714 : BOOL; (*measuring signal failure return water temperature primary circuit*) (*OldName:newPv; Cycle:5;*)
		bMsg2715 : BOOL; (*measuring signal failure supply water temperature secondary circuit*) (*OldName:newPv; Cycle:5;*)
		bMsg2716 : BOOL; (*measuring signal failure return water temperature secondary circuit*) (*OldName:newPv; Cycle:5;*)
		bMsg2717 : BOOL; (*supply water temperature high primary circuit*) (*OldName:newPv; Cycle:5;*)
		bMsg2718 : BOOL; (*return water temperature high primary circuit*) (*OldName:newPv; Cycle:5;*)
		bMsg2719 : BOOL; (*supply water temperature high secondary circuit*) (*OldName:newPv; Cycle:5;*)
		bMsg2720 : BOOL; (*return water temperature high secondary circuit*) (*OldName:newPv; Cycle:5;*)
		bMsg2721 : BOOL; (*measuring signal failure heating power engine heat water circuit*) (*OldName:newPv; Cycle:5;*)
		bMsg2731 : BOOL; (*measuring signal failure supply temperature condensor circuit*) (*OldName:newPv; Cycle:5;*)
		bMsg2732 : BOOL; (*supply temperature condensor circuit maximum*) (*OldName:newPv; Cycle:5;*)
		bMsg2733 : BOOL; (*measuring signal failure return temperature condensor circuit*) (*OldName:newPv; Cycle:5;*)
		bMsg2734 : BOOL; (*return temperature condensor circuit maximum*) (*OldName:newPv; Cycle:5;*)
		bMsg2735 : BOOL; (*failure condensor pump*) (*OldName:newPv; Cycle:5;*)
		bMsg2736 : BOOL; (*Failure boiler house ventilation*) (*OldName:newPv; Cycle:5;*)
		bMsg2750 : BOOL; (*failure heat circuit flap*) (*OldName:newPv; Cycle:5;*)
		bMsg2751 : BOOL; (*heat circuit return temperature high*) (*OldName:newPv; Cycle:5;*)
		bMsg2752 : BOOL; (*signal failure heat circuit return temperature high*) (*OldName:newPv; Cycle:5;*)
		bMsg2763 : BOOL; (*plausibility check measuring signal engine cooling water pressure*)
		bMsg3220 : BOOL; (*engine cooling water temperature high*) (*OldName:AMM_W32xx[]; Cycle:5;*)
		bMsg3303 : BOOL; (*signal failure heat water return temp. after EC trip*) (*OldName:AMM_A33xx[]; Cycle:5;*)
		bMsg3312 : BOOL; (*signal failure heat water return temp. after EC trip*) (*OldName:AMM_A33xx[]; Cycle:5;*)
		bMsg3321 : BOOL; (*signal failure heat  water return temperature trip*) (*OldName:AMM_A33xx[]; Cycle:5;*)
		bMsg3402 : BOOL; (*engine cooling water pressure low*) (*OldName:AMM_W34xx[]; Cycle:5;*)
		bMsg3404 : BOOL; (*water pressure cooler circuit low*)
		bMsg3406 : BOOL; (*engine cooling water pressure high*)
		bMsg3407 : BOOL; (*signal failure outdoor temperature*)
		bMsg3492 : BOOL; (*temperature engine cooling water before charge cooler high temp.circuit active M.06-TI-014*)
		bMsg3493 : BOOL; (*temperature engine cooling water before oil cooler active M.06-TI-020*)
		bMsg3494 : BOOL; (*temperature engine cooling water before engine cooling water cooler active M.06-TI-030*)
		bMsg3508 : BOOL; (*signal failure heat water return temp. after EC*)
		bMsg3509 : BOOL; (*heat water return temperature after EC high*)
		bMsg3521 : BOOL; (*charge cooling water temperature high*)
		bMsg3526 : BOOL; (*signal failure heat  water return temperature before engine*)
		bMsg3527 : BOOL; (*heat water return temperature before engine high*)
		bMsg3590 : BOOL; (*signal failure temp. heat water return low temperatur*)
		bMsg9098 : BOOL; (*Valve heating in operation*)
		bMsg9099 : BOOL; (*Ring heater for cooling fan in operation*)
		bMsg9226 : BOOL; (*charge cooler 2 water pressure low*) (*OldName:newPV; Cycle:5;*)
		bMsg9228 : BOOL; (*charge cooler 2 failure*) (*OldName:newPV; Cycle:5;*)
		bMsg9229 : BOOL; (*Charge cooler 2 water temperature high*) (*OldName:newPV; Cycle:5;*)
		bMsg9230 : BOOL; (*Measuring signal failure position temperature-control-valve charge cooler 2 circuit*) (*OldName:newPV; Cycle:5;*)
		bMsg9231 : BOOL; (*Measuring signal failure supply water temperature charge cooler 2 circuit*) (*OldName:newPV; Cycle:5;*)
		bMsg9232 : BOOL; (*Measuring signal failure return water temperature charge cooler 2 circuit*) (*OldName:newPV; Cycle:5;*)
		bChC_DemPump : BOOL; (*charge cooler demand pump*) (*OldName:GKP_EIN; Cycle:5;*)
		bEC_DemPump : BOOL; (*emergency cooler demand pump*) (*OldName:KP_EIN; Cycle:5;*)
		bChC_Heating_Dem : BOOL; (*Charge cooler pre heating*) (*OldName:FG_KT; Cycle:5;*)
		rT_ECW_bChC_HT : REAL; (*temperature engine cooling water before charge cooler high temp.circ. M.06-TI-014*) (*OldName:newPv; Cycle:5;*)
		rT_ECW_bOilC : REAL; (*temperature engine cooling water before oil cooler M.06-TI-020*) (*OldName:newPv; Cycle:5;*)
		rT_ECW_bECWC : REAL; (*temperature engine cooling water before engine cooling water cooler M.06-TI-030*) (*OldName:newPv; Cycle:5;*)
		bEC_On : BOOL; (*emergency cooler on*) (*OldName:newPv; Cycle:5;*)
		bChC_On : BOOL; (*charge cooler on*) (*OldName:newPv; Cycle:5;*)
		bChC2_DemPump : BOOL; (*charge cooler 2 demand pump*) (*OldName:newPV; Cycle:5;*)
		tCtr_ChC_T1HP_Out : _tGeACtrOut; (*charge temperature before high-pressure turbo charger controller*) (*OldName:newPV; Cycle:5;*)
		rPos_ChC2_Valve : REAL; (*Position temperature-regulation-valve 2nd LT charge cooler circuit (T1-HP)*) (*OldName:newPv; Cycle:5;*)
		iSumChC2_Stages : INT; (*summary charge cooler 2 stages*) (*OldName:newPV; Cycle:5;*)
		bChC2_On : BOOL; (*charge cooler 2 on*) (*OldName:newPv; Cycle:5;*)
		bChC2_Heating_Dem : BOOL; (*Charge cooler 2 pre heating*) (*OldName:newPV; Cycle:5;*)
		rT_ChC2_Su_LT : REAL; (*supply water temperature charge cooler 2 [°C]*) (*OldName:newPV; Cycle:5;*)
		rT_ChC2_Re_LT : REAL; (*return water temperature charge cooler 2 [°C]*) (*OldName:newPV; Cycle:5;*)
		bECW_ShutOffVal_Dem : BOOL; (*demand 2-way shut off valve engine jacket water circuit*)
		bECW_ShutOffVal_Dem_Exist : BOOL; (*demand 2-way shut off valve engine jacket water circuit exist*)
		bValHeater_Dem : BOOL; (*demand 3-way valve heater*)
		bValHeater_Dem_Exist : BOOL; (*demand 3-way valve heater exist*)
		bFanRingHeater_Dem : BOOL; (*demand fan ring heater*)
		bFanRingHeater_Dem_Exist : BOOL; (*demand fan ring heater exist*)
		rT_HW_Su_Unit : REAL; (*SAFETY PLC: Heating water supply temperature - Unit (M.06-TI-003)*) (*OldName: new PV; Cycle: 5;*) (*V04.25.00.00*)
		bMsg9588 : BOOL; (*SAFETY PLC: Heating water supply temperature unit maximum*) (*OldName: new PV; Cycle: 5;*) (*V04.25.00.00*)
		bMsg9589 : BOOL; (*SAFETY PLC: Heating water supply temperature unit measuring signal failure*) (*OldName: new PV; Cycle: 5;*) (*V04.25.00.00*)
	END_STRUCT; (*END_MM2VIS*)
	tManAuxCtr_typ : 	STRUCT
		bGnl_Rel : BOOL; (*General release. Safety conditions (gas alarm, fire alarm, safety loop, ..) are OK.*) (*OldName: new PV; Cycle: 5;*)
		bECWP_PreH_COf_Man : BOOL; (*engine cooling water pump preheating demand off*) (*OldName: new PV; Cycle: 5;*)
		bECW_PreH_COf_Man : BOOL; (*engine cooling water preheating demand off*) (*OldName: new PV; Cycle: 5;*)
		bInAirER_Lou2DemOpen_Man : BOOL; (*demand open air inlet louver 2*) (*OldName: new PV; Cycle:5;*)
		bInAirER_Lou1DemOpen_Man : BOOL; (*demand open air inlet louver 1*) (*OldName: new PV; Cycle:5;*)
		bOutAirER_LouDemOpen_Man : BOOL; (*open air outlet louver *) (*OldName: new PV; Cycle:5;*)
		bInAirER_Fan1DemOn_Man : BOOL; (*demand air inlet ventilator 1*) (*OldName: new PV; Cycle:5;*)
		bInAirER_Fan2DemOn_Man : BOOL; (*demand air inlet ventilator 2*) (*OldName: new PV; Cycle:5;*)
		bER_FC_Set_Man : BOOL; (*demand engine room frequency converter setpoint*) (*OldName: new PV; Cycle:5;*)
		rER_FC_Set_Man : REAL; (*engine room frequency converter setpoint [%]*) (*OldName: new PV; Cycle:5;*)
		bER_OutlV_FC_Set_Man : BOOL; (*demand engine room air outlet ventilation frequency converter setpoint*) (*OldName: new PV; Cycle:5;*)
		rER_OutlV_FC_Set_Man : REAL; (*engine room air outlet ventilation frequency converter setpoint [%]*) (*OldName: new PV; Cycle:5;*)
		bEC_DemPump_Man : BOOL; (*emergency cooler demand pump*) (*OldName: new PV; Cycle:5;*)
		bEC_DemFan_Man : BOOL; (*emergency cooler demand fan 1 - 16*) (*OldName: new PV; Cycle:5;*)
		bChC_DemPump_Man : BOOL; (*charge cooler demand pump*) (*OldName: new PV; Cycle:5;*)
		bChC_DemFan_Man : BOOL; (*charge cooler demand fan 1 - 16*) (*OldName: new PV; Cycle:5;*)
		bEG_BoVaCoOpen_Man : BOOL; (*exhaust gas boiler valve command open*) (*OldName: new PV; Cycle:5;*)
		bEG_BoVaCoClose_Man : BOOL; (*exhaust gas boiler valve command close*) (*OldName: new PV; Cycle:5;*)
		bEG_ByVaCoOpen_Man : BOOL; (*exhaust gas bypass valve command open*) (*OldName: new PV; Cycle:5;*)
		bEG_ByVaCoClose_Man : BOOL; (*exhaust gas bypass valve command close*) (*OldName: new PV; Cycle:5;*)
		bAuxCust_Man : ARRAY[0..40]OF BOOL; (*reserve customer auxiliaries*) (*OldName: new PV; Cycle:5;*)
		bCDP_Dem_Man : BOOL; (*demand condensor pump*) (*OldName: new PV; Cycle:5;*)
		bBHV_Dem_Man : BOOL; (*demand boiler house ventilation*) (*OldName: newPv; Cycle:5;*)
		bHWF_Dem_Man : BOOL; (*demand heating circuit flap*) (*OldName:newPv; Cycle:5;*)
		bChC_Heating_Man : BOOL; (*charge cooler pre heating*) (*OldName:newPv; Cycle:5;*)
		bCO2_DemCodinox_Man : BOOL; (*CO2 demand CODINOX*) (*OldName:newPv; Cycle:5;*)
		bECWP_PreH_COf : BOOL; (*engine cooling water pump preheating demand off*) (*OldName: new PV; Cycle: 5;*)
		bECW_PreH_COf : BOOL; (*engine cooling water preheating demand off*) (*OldName: new PV; Cycle: 5;*)
		bInAirER_Lou2DemOpen : BOOL; (*demand open air inlet louver 2*) (*OldName: new PV; Cycle:5;*)
		bInAirER_Lou1DemOpen : BOOL; (*demand open air inlet louver 1*) (*OldName: new PV; Cycle:5;*)
		bOutAirER_LouDemOpen : BOOL; (*open air outlet louver *) (*OldName: new PV; Cycle:5;*)
		bInAirER_Fan1DemOn : BOOL; (*demand air inlet ventilator 1*) (*OldName: new PV; Cycle:5;*)
		bInAirER_Fan2DemOn : BOOL; (*demand air inlet ventilator 2*) (*OldName: new PV; Cycle:5;*)
		bER_OutlV_FC_Set : BOOL; (*demand engine room air outlet ventilation frequency converter setpoint*) (*OldName: new PV; Cycle:5;*)
		rER_OutlV_FC_Set : REAL; (*engine room air outlet ventilation frequency converter setpoint [%]*) (*OldName: new PV; Cycle:5;*)
		bER_FC_Set : BOOL; (*demand engine room frequency converter setpoint*) (*OldName: new PV; Cycle:5;*)
		rER_FC_Set : REAL; (*engine room frequency converter setpoint [%]*) (*OldName: new PV; Cycle:5;*)
		bEC_DemPump : BOOL; (*emergency cooler demand pump*) (*OldName: new PV; Cycle:5;*)
		bEC_DemFan : BOOL; (*emergency cooler demand fan 1 - 16*) (*OldName: new PV; Cycle:5;*)
		bChC_DemPump : BOOL; (*charge cooler demand pump*) (*OldName: new PV; Cycle:5;*)
		bChC_DemFan : BOOL; (*charge cooler demand fan 1 - 16*) (*OldName: new PV; Cycle:5;*)
		bEG_BoVaCoOpen : BOOL; (*exhaust gas boiler valve command open*) (*OldName: new PV; Cycle:5;*)
		bEG_BoVaCoClose : BOOL; (*exhaust gas boiler valve command close*) (*OldName: new PV; Cycle:5;*)
		bEG_ByVaCoOpen : BOOL; (*exhaust gas bypass valve command open*) (*OldName: new PV; Cycle:5;*)
		bEG_ByVaCoClose : BOOL; (*exhaust gas bypass valve command close*) (*OldName: new PV; Cycle:5;*)
		bAuxCust : ARRAY[0..70]OF BOOL; (*reserve customer auxiliaries*) (*OldName: new PV; Cycle:5;*)
		bCDP_Dem : BOOL; (*demand condensor pump*) (*OldName: new PV; Cycle:5;*)
		bBHV_Dem : BOOL; (*demand boiler house ventilation*) (*OldName: newPv; Cycle:5;*)
		bHWF_Dem : BOOL; (*demand heating circuit flap*) (*OldName:newPv; Cycle:5;*)
		bChC_Heating : BOOL; (*charge cooler pre heating*) (*OldName:newPv; Cycle:5;*)
		bCO2_DemCodinox : BOOL; (*CO2 demand CODINOX*) (*OldName:newPv; Cycle:5;*)
		bChC2_DemPump : BOOL; (*charge cooler 2 demand pump*) (*OldName: new PV; Cycle:5;*)
		bChC2_DemPump_Man : BOOL; (*charge cooler 2 demand pump*) (*OldName: new PV; Cycle:5;*)
		bChC2_DemFan : BOOL; (*charge cooler 2 demand fan 1 - 16*) (*OldName: new PV; Cycle:5;*)
		bChC2_DemFan_Man : BOOL; (*charge cooler 2 demand fan 1 - 16*) (*OldName: new PV; Cycle:5;*)
		bChC2_Heating : BOOL; (*charge cooler 2 pre heating*) (*OldName:newPv; Cycle:5;*)
		bChC2_Heating_Man : BOOL; (*charge cooler 2 pre heating*) (*OldName:newPv; Cycle:5;*)
		bECW_HydrPreH_COf : BOOL; (*engine cooling water hydraulic preheating demand off*) (*OldName: new PV; Cycle: 5;*)
		bECW_HydrPreH_COf_Man : BOOL; (*engine cooling water hydraulic preheating demand off*) (*OldName: new PV; Cycle: 5;*)
		bEOP_DemPump : BOOL; (*engine prelubrication pump manual demand*) (*OldName: new PV; Cycle: 5;*)
		bEOP_DemPump_Man : BOOL; (*engine prelubrication pump manual demand*) (*OldName: new PV; Cycle: 5;*)
	END_STRUCT;
	Perm_HC_Struct : 	STRUCT
		iCnt_P_Heat : DINT; (*heat counter*)
		rPermValue01 : REAL; (*spare permanent value - replace with new vars of same lenght, when needed*)
		rPermValue02 : REAL; (*spare permanent value - replace with new vars of same lenght, when needed*)
		rPermValue03 : REAL; (*spare permanent value - replace with new vars of same lenght, when needed*)
		rPermValue04 : REAL; (*spare permanent value - replace with new vars of same lenght, when needed*)
		rPermValue05 : REAL; (*spare permanent value - replace with new vars of same lenght, when needed*)
		rPermValue06 : REAL; (*spare permanent value - replace with new vars of same lenght, when needed*)
		rPermValue07 : REAL; (*spare permanent value - replace with new vars of same lenght, when needed*)
		rPermValue08 : REAL; (*spare permanent value - replace with new vars of same lenght, when needed*)
		rPermValue09 : REAL; (*spare permanent value - replace with new vars of same lenght, when needed*)
		rPermValue10 : REAL; (*spare permanent value - replace with new vars of same lenght, when needed*)
	END_STRUCT;
END_TYPE
```

### module_HCPara.typ - Local data types
```iecst
TYPE
	PROGRAMMER_INFO : 	STRUCT
		DO_NOT_SORT_PARA : STRING[40] := 'DO NOT CHANGE PARAMETER SORTING!'; (*DO NOT CHANGE PARAMETER SORTING!*) (*ADD NEW PARAMETER ONLY AT THE END OF THE Para STRUCTURE. DO NOT DELETE existing Para items.*)
	END_STRUCT;
	PARA_HC_Struct : 	STRUCT  (*! Add new tags only at the end OF the pm structure!*)
		tCtr_Cust1 : _tGeACtrPara; (*Para controller customized*) (*OldName:bTuneREG1_Invert; Cycle:5;*)
		tCtr_Cust2 : _tGeACtrPara; (*Para controller customized*) (*OldName:bTuneREG2_Invert; Cycle:5;*)
		tCtr_Cust3 : _tGeACtrPara; (*Para controller customized*) (*OldName:bTuneREG3_Invert; Cycle:5;*)
		tCtr_Cust4 : _tGeACtrPara; (*Para controller customized*) (*OldName:bTuneREG4_Invert; Cycle:5;*)
		tCtr_Cust5 : _tGeACtrPara; (*Para controller customized*) (*OldName:bTuneREG5_Invert; Cycle:5;*)
		tCtr_Cust6 : _tGeACtrPara; (*Para controller customized*) (*OldName:bTuneREG6_Invert; Cycle:5;*)
		tCtr_Cust7 : _tGeACtrPara; (*Para controller customized*) (*OldName:bTuneREG7_Invert; Cycle:5;*)
		tCtr_Cust8 : _tGeACtrPara; (*Para controller customized*) (*OldName:bTuneREG8_Invert; Cycle:5;*)
		tCtr_EC : _tGeACtrPara; (*Para controller emergency cooler*) (*OldName:REG11; Cycle:5;*)
		tCtr_HWRe : _tGeACtrPara; (*Para controller heat water return temperature*) (*OldName:REG10; Cycle:5;*)
		tCtr_HWSu : _tGeACtrPara; (*Para controller heat water supply temperature*) (*OldName:REG14; Cycle:5;*)
		tCtr_ChCHP : _tGeACtrPara; (*Para controller charge temperature cooler high pressure*) (*OldName:REG18; Cycle:5;*)
		tCtr_ChCV : _tGeACtrPara; (*Para controller charge temperature  cooler ventilation*) (*OldName:REG15; Cycle:5;*)
		tCtr_ChC : _tGeACtrPara; (*Para controller charge temperature cooler*) (*OldName:REG9; Cycle:5;*)
		rN_EngStart_LimHi : REAL; (*PARA [11296]: engine start speed limit high [1/min]*) (*OldName:GW_DREHZ; Cycle:5;*)
		rN_EngStart_HyHi : REAL; (*PARA [11295]: engine start speed limit high hysteresis [1/min]*) (*OldName:HY_DREHZ; Cycle:5;*)
		bCtr_ChC : BOOL; (*PARA [11872]: visibility charge temperature controller*) (*OldName:bPlantCtr9,reg0_visible; Cycle:5;*)
		bCtr_ChCV : BOOL; (*PARA [11874]: visibility charge cooler ventilation controller*) (*OldName:bPlantCtr15; Cycle:5;*)
		bCtr_ChCHP : BOOL; (*PARA [11873]: visibility charge temperature controller, high pressure*) (*OldName:bPlantCtr18; Cycle:5;*)
		bCtr_EC : BOOL; (*PARA [11875]: visibility emergency controller(dump radiator)*) (*OldName:bPlantCtr11; Cycle:5;*)
		bCtr_HWRe : BOOL; (*PARA [11876]: visibility heat water return temperature controller*) (*OldName:bPlantCtr10; Cycle:5;*)
		bCtr_HWSu : BOOL; (*PARA [11877]: visibility heat water supply temperature controller*) (*OldName:bPlantCtr14; Cycle:5;*)
		iEng_Motortype : INT; (*Para engine type*) (*OldName:motortyp; Cycle:5;*)
		bT_HW_Su_SF_Trip : BOOL; (*PARA [11893]: temperature heat water supply signal failure trip*) (*OldName:vorl_msa; Cycle:5;*)
		bT_HW_Re_SF_Trip : BOOL; (*PARA [11887]: temperature heat water  return signal failure trip*) (*OldName:rueckl_msa; Cycle:5;*)
		bT_HW_ReAfEC_SF_Trip : BOOL; (*PARA [11889]: temperature heat water  return after EC signal failure trip*) (*OldName:rlt_nk_msa; Cycle:5;*)
		bVISA : BOOL; (*PARA [12259]: monitoring acc. VISA*) (*OldName:VISA; Cycle:5;*)
		rT_AirOutdoor_LimHi2 : REAL; (*PARA [11927]: temperature air outdoor limit high [°C]*) (*OldName:GW_ULT_2; Cycle:5;*)
		rT_AirOutdoor_LimHi3 : REAL; (*PARA [11928]: temperature air outdoor limit high [°C]*) (*OldName:GW_ULT_3; Cycle:5;*)
		rT_AirOutdoor_LimHi4 : REAL; (*PARA [11929]: temperature air outdoor limit high [°C]*) (*OldName:GW_ULT_4; Cycle:5;*)
		rT_AirOutdoor_LimHi1 : REAL; (*PARA [11926]: temperature air outdoor limit high [°C]*) (*OldName:GW_ULT_1; Cycle:5;*)
		rT_AirOutdoor_HyHi2 : REAL; (*PARA [11923]: temperature air outdoor hysteres limit high [°C]*) (*OldName:HY_ULT_2; Cycle:5;*)
		rT_AirOutdoor_HyHi3 : REAL; (*PARA [11924]: temperature air outdoor hysteres limit high [°C]*) (*OldName:HY_ULT_3; Cycle:5;*)
		rT_AirOutdoor_HyHi4 : REAL; (*PARA [11925]: temperature air outdoor hysteres limit high [°C]*) (*OldName:HY_ULT_4; Cycle:5;*)
		rT_AirOutdoor_HyHi1 : REAL; (*PARA [11922]: temperature air outdoor hysteres limit high [°C]*) (*OldName:HY_ULT_1; Cycle:5;*)
		iEC_NumDemAux : INT; (*PARA [11899]: number emergency cooler stages with demand auxiliaries*) (*OldName:Anz_hbt; Cycle:5;*)
		iEC_NumStages : INT; (*PARA [11900]: emergency cooler number of cooling steps total*) (*OldName:K_anz; Cycle:5;*)
		iChC_NumDemAux : INT; (*PARA [11895]: number charge cooler stages with demand auxiliaries*) (*OldName:Anz_GK_hbt; Cycle:5;*)
		iChC_NumStages : INT; (*PARA [11896]: charge cooler number stages*) (*OldName:GK_anz; Cycle:5;*)
		iChC_OpMode : INT; (*PARA [11897]: charge cooler operating mode*) (*OldName:GK_var; Cycle:5;*)
		iChC_CtrNum : INT; (*PARA [11894]: charge cooler controller number*) (*OldName:GK_reg; Cycle:5;*)
		bEC_St1onlyP : BOOL; (*PARA [11879]: emergency cooler first stage only with pump*) (*OldName:K_nmp; Cycle:5;*)
		rEC_ValPosLimHi_On : REAL; (*PARA [11909]: emergency cooler activation from  valve position limit high [%]*) (*OldName:GW_K_EIN; Cycle:5;*)
		rPr_ECW_LimLo1 : REAL; (*PARA [11918]: pressure engine cooling water limit low 1 [bar]*) (*OldName:GW_KDGW1; Cycle:5;*)
		rPr_ECW_LimHiHi : REAL; (*PARA [11916]: pressure engine cooling water limit high high [bar]*) (*OldName:GW_KDMA; Cycle:5;*)
		rPr_ECW_LimLoLo : REAL; (*PARA [11919]: pressure engine cooling water limit low low [bar]*) (*OldName:GW_KDMI; Cycle:5;*)
		rPr_ECW_LimLo : REAL; (*PARA [11917]: pressure engine cooling water limit low [bar]*) (*OldName:GW_KDMI_W; Cycle:5;*)
		rT_ECW_LimHi1 : REAL; (*PARA [11942]: temperature engine cooling water limit high 1 [°C]*) (*OldName:GW_KTGW1; Cycle:5;*)
		rT_ECW_LimHi2 : REAL; (*PARA [11943]: temperature engine cooling water limit high 2 [°C]*) (*OldName:GW_KTGW2; Cycle:5;*)
		rT_ECW_LimHi : REAL; (*PARA [11941]: temperature engine cooling water limit high [°C]*) (*OldName:GW_KTMA; Cycle:5;*)
		rT_ECW_LimLo : REAL; (*PARA [11944]: temperature engine cooling water limit low [°C]*) (*OldName:GW_KTMI; Cycle:5;*)
		rT_ECW_LimRelLoad : REAL; (*PARA [11945]: temperature engine cooling water limit release load [°C]*) (*OldName:GW_LFG; Cycle:5;*)
		rEC_ValPosLimStageDown : REAL; (*PARA [11910]: position emergency cooler valve limit stage down [%]*) (*OldName:GW_MINUS; Cycle:5;*)
		rEC_ValPosLimStageUp : REAL; (*PARA [11911]: position emergency cooler valve limit stage up [%]*) (*OldName:GW_PLUS; Cycle:5;*)
		rT_HW_ReBeEng_LimHi : REAL; (*PARA [11960]: temperature heat water return before engine limit high [°C]*) (*OldName:GW_RLT_M; Cycle:5;*)
		rT_HW_ReBeEng_LimHiHi : REAL; (*PARA [11961]: temperature heat water return before engine limit high high [°C]*) (*OldName:GW_RLT_MA; Cycle:5;*)
		rT_HW_ReAfEC_LimHi : REAL; (*PARA [11956]: temperature heat water return after emergency cooler limit high [°C]*) (*OldName:GW_RLT_NK; Cycle:5;*)
		rT_HW_ReAfEC_LimHiHi : REAL; (*PARA [11957]: temperature heat water return after emergency cooler limit high high [°C]*) (*OldName:GW_RLT_NKA; Cycle:5;*)
		rT_HW_Re_LimHi : REAL; (*PARA [11952]: temperature heat water return limit high [°C]*) (*OldName:GW_RLTP; Cycle:5;*)
		rT_HW_Re_LimHiHi : REAL; (*PARA [11953]: temperature heat water return limit high high [°C]*) (*OldName:GW_RLTPA; Cycle:5;*)
		rT_HW_Su_LimHi : REAL; (*PARA [11964]: temperature heat water supply limit high [°C]*) (*OldName:GW_VLTP; Cycle:5;*)
		rT_HW_Su_LimHiHi : REAL; (*PARA [11965]: temperature heat water supply limit high high [°C]*) (*OldName:GW_VLTPA; Cycle:5;*)
		rT_ECW_PreH_LimOFF : REAL; (*PARA [10089]: temperature engine cooling water preheating limit off [°C]*) (*OldName:GW_VORW; Cycle:5;*)
		rEC_ValPosHyHi_On : REAL; (*PARA [11908]: position valve emergency cooler ON limit high hysteresis [%]*) (*OldName:HY_K_EIN; Cycle:5;*)
		rPr_ECW_HyLo1 : REAL; (*PARA [11914]: pressure engine cooling water limit low 1 hysteresis [bar]*) (*OldName:HY_KDGW1; Cycle:5;*)
		rPr_ECW_HyHiHi : REAL; (*PARA [11912]: pressure engine cooling water limit high high hysteresis [bar]*) (*OldName:HY_KDMA; Cycle:5;*)
		rPr_ECW_HyLoLo : REAL; (*PARA [11915]: pressure engine cooling water limit low low hysteresis [bar]*) (*OldName:HY_KDMI; Cycle:5;*)
		rPr_ECW_HyLo : REAL; (*PARA [11913]: pressure engine cooling water limit low hysteresis [bar]*) (*OldName:HY_KDMI_W; Cycle:5;*)
		rT_ECW_HyHi1 : REAL; (*PARA [11936]: temperature engine cooling water limit high 1 hysteresis [°C]*) (*OldName:HY_KTGW1; Cycle:5;*)
		rT_ECW_HyHi2 : REAL; (*PARA [11937]: temperature engine cooling water limit high 2 hysteresis [°C]*) (*OldName:HY_KTGW2; Cycle:5;*)
		rT_ECW_HyHi : REAL; (*PARA [11935]: temperature engine cooling water limit high hysteresis [°C]*) (*OldName:HY_KTMA; Cycle:5;*)
		rT_ECW_HyLo : REAL; (*PARA [11938]: temperature engine cooling water limit low hysteresis [°C]*) (*OldName:HY_KTMI; Cycle:5;*)
		rT_ECW_HyRelLoad : REAL; (*PARA [11939]: temperature engine cooling water limit release load hysteresis [°C]*) (*OldName:HY_LFG; Cycle:5;*)
		rT_HW_ReBeEng_HyHi : REAL; (*PARA [11958]: temperature heat water return before engine limit high hysteresis [°C]*) (*OldName:HY_RLT_M; Cycle:5;*)
		rT_HW_ReBeEng_HyHiHi : REAL; (*PARA [11959]: temperature heat water return before engine limit high high hysteresis [°C]*) (*OldName:HY_RLT_MA; Cycle:5;*)
		rT_HW_ReAfEC_HyHi : REAL; (*PARA [11954]: temperature heat water return after emergency cooler limit high hysteresis [°C]*) (*OldName:HY_RLT_NK; Cycle:5;*)
		rT_HW_ReAfEC_HyHiHi : REAL; (*PARA [11955]: temperature heat water return after emergency cooler limit high high hysteresis [°C]*) (*OldName:HY_RLT_NKA; Cycle:5;*)
		rT_HW_Re_HyHi : REAL; (*PARA [11950]: temperature heat water return limit high hysteresis [°C]*) (*OldName:HY_RLTP; Cycle:5;*)
		rT_HW_Re_HyHiHi : REAL; (*PARA [11951]: temperature heat water return limit high high hysteresis [°C]*) (*OldName:HY_RLTPA; Cycle:5;*)
		rT_HW_Su_HyHi : REAL; (*PARA [11962]: temperature heat water supply limit high hysteresis [°C]*) (*OldName:HY_VLTP; Cycle:5;*)
		rT_HW_Su_HyHiHi : REAL; (*PARA [11963]: temperature heat water supply limit high high hysteresis [°C]*) (*OldName:HY_VLTPA; Cycle:5;*)
		rT_ECW_PreH_HyOFF : REAL; (*PARA [10088]: temperature engine cooling water preheating limit off hysteresis [°C]*) (*OldName:HY_VORW; Cycle:5;*)
		iEC_NumCtr : INT; (*PARA [11898]: emergency cooler number of PLC controller for valve control*) (*OldName:K_reg; Cycle:5;*)
		iEC_OpMode : INT; (*PARA [11901]: emergency cooler operating mode selection*) (*OldName:K_var; Cycle:5;*)
		bT_HW_ReBeEng_Active : BOOL; (*PARA [11890]: temperature heat water return before engine measurement active*) (*OldName:rlt_m_a; Cycle:5;*)
		bT_HW_ReBeEng_SF_Trip : BOOL; (*PARA [11891]: temperature heat water return before engine signal failure trip*) (*OldName:rlt_msa_a; Cycle:5;*)
		bT_HW_ReAfEC_Active : BOOL; (*PARA [11888]: temperature heat water return after emergency cooler measurement active*) (*OldName:rlt_nk_a; Cycle:5;*)
		bT_HW_Re_Active : BOOL; (*PARA [11886]: temperature heat water return measurement active*) (*OldName:rueckl_a; Cycle:5;*)
		tiEC_DelayOff : TIME; (*PARA [12050]: emergency cooler delay OFF*) (*OldName:TW_K_AUS; Cycle:5;*)
		tiEC_DelayStageDown : TIME; (*PARA [12051]: emergency cooler delay switch stage down*) (*OldName:TW_MINUS; Cycle:5;*)
		tiEC_DelayStageUp : TIME; (*PARA [12052]: emergency cooler delay switch stage up*) (*OldName:TW_PLUS; Cycle:5;*)
		bT_AirOutdoor_Active : BOOL; (*PARA [11885]: air outdoor temperature measurement enable *) (*OldName:ULT_a; Cycle:5;*)
		bT_HW_Su_Active : BOOL; (*PARA [11892]: temperature heat water supply measurement active*) (*OldName:vorl_a; Cycle:5;*)
		rT_Ch_LimHi1 : REAL; (*PARA [11932]: charge temperature high limit 1 [°C]*) (*OldName:GW_LLGW1; Cycle:5;*)
		rT_Ch_LimHi2 : REAL; (*PARA [11933]: charge temperature high limit 2 [°C]*) (*OldName:GW_LLGW2; Cycle:5;*)
		rT_Ch_HyHi1 : REAL; (*PARA [11930]: charge temperature high hysteresis limit 1 [°C]*) (*OldName:HY_LLGW1; Cycle:5;*)
		rT_Ch_HyHi2 : REAL; (*PARA [11931]: charge temperature high hysteresis limit 2 [°C]*) (*OldName:HY_LLGW2; Cycle:5;*)
		rT_EO_LimHi2 : REAL; (*PARA [11949]: engine oil temperature high limit 2 [°C]*) (*OldName:GW_OTGW2; Cycle:5;*)
		rT_EO_LimHi1 : REAL; (*PARA [11948]: engine oil temperature high limit 1 [°C]*) (*OldName:GW_OTGW1; Cycle:5;*)
		rT_EO_HyHi2 : REAL; (*PARA [11947]: engine oil temperature high hysteresis limit 2 [°C]*) (*OldName:HY_OTGW2; Cycle:5;*)
		rT_EO_HyHi1 : REAL; (*PARA [11946]: engine oil temperature high hysteresis limit 1 [°C]*) (*OldName:HY_OTGW1; Cycle:5;*)
		rChC_ValPosLimHi_On : REAL; (*PARA [11905]: position valve charge cooler ON limit high [%]*) (*OldName:GW_GK_EIN; Cycle:5;*)
		rChC_ValPosHyHi_On : REAL; (*PARA [11904]: position valve charge cooler ON limit high hysteresis [%]*) (*OldName:HY_GK_EIN; Cycle:5;*)
		rChC_ValPosLimStageUp : REAL; (*PARA [11907]: position charge cooler valve limit stage up [%]*) (*OldName:GW_GK_PLUS; Cycle:5;*)
		rChC_ValPosLimStageDown : REAL; (*PARA [11906]: position charge cooler valve limit stage down [%]*) (*OldName:GW_GK_MINUS; Cycle:5;*)
		tiChC_DelayOff : TIME; (*PARA [12047]: charge cooler delay OFF*) (*OldName:TW_GK_AUS; Cycle:5;*)
		tiChC_DelayStageUp : TIME; (*PARA [12049]: charge cooler delay switch stage up *) (*OldName:TW_GK_PLUS; Cycle:5;*)
		tiChC_DelayStageDown : TIME; (*PARA [12048]: charge cooler delay switch stage down*) (*OldName:TW_GK_MINUS; Cycle:5;*)
		iPred_T_HW_Re_Sel : INT; (*PARA [11903]: power reduction heat water return temperature high active*) (*OldName:Pred_RLT_act; Cycle:5;*)
		rT_Pred_HW_Re_Start : REAL; (*PARA [11967]: power reduction heat water return temperature high start [°C]*) (*OldName:Pred_RLT_start; Cycle:5;*)
		rPred_T_HW_Re_Rate : REAL; (*PARA [11921]: power reduction heat water return temperature high rate [%/°C]*) (*OldName:Pred_RLT_rate; Cycle:5;*)
		rT_Pred_ECW_Start : REAL; (*PARA [11966]: power reduction engine cooling water temperature high start [°C]*) (*OldName:Pred_KWT_start; Cycle:5;*)
		rPred_ECW_Rate : REAL; (*PARA [11920]: power reduction engine cooling water temperature high rate [%/°C]*) (*OldName:Pred_KWT_rate; Cycle:5;*)
		bAuxEC_Visible : BOOL; (*PARA [11870]: visibility parameters of emergency cooler control*) (*OldName:bAuxilAirCool; Cycle:5;*)
		bEC_St1_Visible : BOOL; (*PARA [11878]: emergency cooler stage 1 visible*) (*OldName:bCoolRadStage1; Cycle:5;*)
		bEC_St2_Visible : BOOL; (*PARA [11880]: emergency cooler stage 2 visible*) (*OldName:bCoolRadStage2; Cycle:5;*)
		bEC_StX_Visible : BOOL; (*PARA [11881]: emergency cooler stage 0-x visible*) (*OldName:bCoolRadStageX; Cycle:5;*)
		bChC_StX_Visible : BOOL; (*PARA [11871]: charge cooler stage0-x visible*) (*OldName:bMixCoolRadStageX; Cycle:5;*)
		bECW_Circuit_Visible : BOOL; (*PARA [11883]: engine cooling water circuit visible*) (*OldName:bVisuCoolCircuit; Cycle:5;*)
		bEC_Visible : BOOL; (*PARA [11882]: graphic for emergency cooler in HYD diagram visible*) (*OldName:bVisuDeskCooler; Cycle:5;*)
		bECW_PreH_Ext_Visible : BOOL; (*PARA [11884]: bypass to 3-way-thermostatic valve visible*) (*OldName:bVisuExtHeating; Cycle:5;*)
		iECW_PreH_Int_Visible : INT; (*PARA [11902]: engine cooling water preheating device visible*) (*OldName:usVisuIntHeating; Cycle:5;*)
		bT_HW_Re_LT_Active : BOOL; (*PARA [12451]: temperature heat water return low temp.circuit measurement active*) (*OldName:bT_HWR_LT_Active; Cycle:5;*)
		rT_HW_Re_LT_LimHi : REAL; (*PARA [12452]: temperature heat water return low temp.circuit limit high [°C]*) (*OldName:newPv; Cycle:5;*)
		rT_HW_Re_LT_HyHi : REAL; (*PARA [12453]: temperature heat water return low temp.circuit limit high hysteresis [°C]*) (*OldName:newPv; Cycle:5;*)
		rT_ECW_LimBpV : REAL; (*PARA [11940]: temperature engine cooling water bypass valve [°C]*) (*OldName:newPv; Cycle:5;*)
		rT_ECW_HyBpV : REAL; (*PARA [11934]: temperature engine cooling water bypass valve hysteresis [°C]*) (*OldName:newPv; Cycle:5;*)
		rT_T2_Set : ARRAY[0..4]OF REAL; (*PARA [11195], [11196], [11197], [11198]: setpoint charge temperature [°C]*) (*OldName:tg_soll[0..4]; Cycle:5;*)
		bAuxChC_Visible : BOOL; (*PARA [11869]: visibility parameters of charge cooler control*) (*OldName:newPv; Cycle:5;*)
		bT_ECWbEng_Active : BOOL; (*PARA [12741]: engine cooling water temperature before engine measurement active M.04-TI-002*) (*OldName:newPv; Cycle:5;*)
		bPr_ECWaEng_Active : BOOL; (*PARA [12739]: engine cooling water pressure after engine measurement active*) (*OldName:newPv; Cycle:5;*)
		bPr_HW_Su_LT_Active : BOOL; (*PARA [12616]: pressure heat water supply low temp.circuit measurement active*) (*OldName:newPv; Cycle:5;*)
		bPr_HW_Su_HT_Active : BOOL; (*PARA [12645]: pressure heat water supply high temp.circuit measurement active*) (*OldName:newPv; Cycle:5;*)
		bT_HW_Su_LT_Active : BOOL; (*PARA [12647]: temperature heat water supply low temp.circuit measurement active*) (*OldName:newPv; Cycle:5;*)
		bPr_HW_Re_LT_Active : BOOL; (*PARA [12892]: pressure heat water return low temp.circuit measurement active M.07-PI-002*) (*OldName:newPv; Cycle:5;*)
		bPr_HW_Re_HT_Active : BOOL; (*PARA [12895]: pressure heat water return high temp.circuit measurement active M.06-PI-002*) (*OldName:newPv; Cycle:5;*)
		bPr_HW_Re_PreH_ECW_Active : BOOL; (*PARA [12898]: pressure heat water return preheating engine cooling water measurement activ M.04-PI-005 *) (*OldName:newPv; Cycle:5;*)
		bPr_HW_Re_PreH_EO_Active : BOOL; (*PARA [12901]: pressure heat water return preheating engine oil measurement active M.03-PI-005*) (*OldName:newPv; Cycle:5;*)
		bPr_EO_Mod_Out_Active : BOOL; (*PARA [12904]: pressure engine oil module outlet measurement active M.03-PI-006*) (*OldName:newPv; Cycle:5;*)
		bT_ECW_Mod_In_Active : BOOL; (*PARA [12908]: temperature engine cooling water, engine cooling water module inlet measurement active M.04-TI-003*) (*OldName:newPv; Cycle:5;*)
		bT_ECW_Mod_Out_Active : BOOL; (*PARA [12909]: temperature engine cooling water, engine cooling water module outlet measurement active M.04-TI-004*) (*OldName:newPv; Cycle:5;*)
		bT_EO_Mod_In_Active : BOOL; (*PARA [12910]: temperature engine oil, oil module inlet measurement active M.03-TI-004*) (*OldName:newPv; Cycle:5;*)
		bT_EO_Mod_Out_Active : BOOL; (*PARA [12911]: temperature engine oil, oil module outlet measurement active M.03-TI-003*) (*OldName:newPv; Cycle:5;*)
		bT_HW_Su_PreH_ECW_Active : BOOL; (*PARA [12912]: temperature heat water supply preheating engine cooling water measurement activ M.04-TI-005 *) (*OldName:newPv; Cycle:5;*)
		bT_HW_Re_PreH_ECW_Active : BOOL; (*PARA [12913]: temperature heat water return preheating engine cooling water measurement activ M.04-TI-006 *) (*OldName:newPv; Cycle:5;*)
		bT_HW_Su_PreH_EO_Active : BOOL; (*PARA [12914]: temperature heat water supply preheating engine oil measurement activ M.03-TI-005 *) (*OldName:newPv; Cycle:5;*)
		bT_HW_Re_PreH_EO_Active : BOOL; (*PARA [12915]: temperature heat water return preheating engine oil measurement activ M.03-TI-006 *) (*OldName:newPv; Cycle:5;*)
		bT_HW_HC_Re_Active : BOOL; (*PARA [13319]: measuring active heat circuit return temperature*) (*OldName:newPv; Cycle:5;*)
		rT_HW_HC_Re_HyHi : REAL; (*PARA [13321]: maximum hysterese heat circuit temperature maximum*) (*OldName:newPv; Cycle:5;*)
		rT_HW_HC_Re_LimHi : REAL; (*PARA [13320]: maximum heat circuit temperature maximum*) (*OldName:newPv; Cycle:5;*)
		bCtr_CDSu : BOOL; (*PARA [13306]: Condensor circuit supply temperature controller*) (*OldName:newPv; Cycle:5;*)
		tCtr_CDSu : _tGeACtrPara; (*Para controller condensor circuit supply temperature*) (*OldName:newPv; Cycle:5;*)
		bT_CD_Re_Active : BOOL; (*PARA [13284]: measuring active return temperature condensor circuit*) (*OldName:newPv; Cycle:5;*)
		rT_CD_Re_HyHi : REAL; (*PARA [13283]: maximum hysterese return temperature condensor circuit*) (*OldName:newPv; Cycle:5;*)
		rT_CD_Re_LimHi : REAL; (*PARA [13282]: maximum return temperature condensor circuit*) (*OldName:newPv; Cycle:5;*)
		bT_CD_Su_Active : BOOL; (*PARA [13281]: measuring active supply temperature condensor circuit*) (*OldName:newPv; Cycle:5;*)
		rT_CD_Su_HyHi : REAL; (*PARA [13280]: maximum hysterese supply temperatur condensor circuit*) (*OldName:newPv; Cycle:5;*)
		rT_CD_Su_LimHi : REAL; (*PARA [13279]: maximum supply temperatur condensor circuit*) (*OldName:newPv; Cycle:5;*)
		bBHV_Active : BOOL; (*PARA [13307]: boiler house flap active*) (*OldName:newPv; Cycle:5;*)
		rT_Su_PriCirc_LimHi : REAL; (*PARA [13156]: supply water temperature high primary circuit [°C]*) (*OldName: new PV   ; Cycle: 5;*)
		rT_Su_PriCirc_HyLimHi : REAL; (*PARA [13157]: supply water temperature high primary circuit hysteresis [°C]*) (*OldName: new PV   ; Cycle: 5;*)
		rT_Re_PriCirc_LimHi : REAL; (*PARA [13159]: return water temperature high primary circuit [°C]*) (*OldName: new PV   ; Cycle: 5;*)
		rT_Re_PriCirc_HyLimHi : REAL; (*PARA [13160]: return water temperature high primary circuit hysteresis [°C]*) (*OldName: new PV   ; Cycle: 5;*)
		rT_Su_SecCirc_LimHi : REAL; (*PARA [13162]: supply water temperature high secondary circuit [°C]*) (*OldName: new PV   ; Cycle: 5;*)
		rT_Su_SecCirc_HyLimHi : REAL; (*PARA [13163]: supply water temperature high secondary circuit hysteresis [°C]*) (*OldName: new PV   ; Cycle: 5;*)
		rT_Re_SecCirc_LimHi : REAL; (*PARA [13165]: return water temperature high secondary circuit [°C]*) (*OldName: new PV   ; Cycle: 5;*)
		rT_Re_SecCirc_HyLimHi : REAL; (*PARA [13166]: return water temperature high secondary circuit hysteresis [°C]*) (*OldName: new PV   ; Cycle: 5;*)
		bT_Su_PriCirc_Active : BOOL; (*PARA [13155]: supply water temperature primary circuit measurement active*) (*OldName: new PV   ; Cycle: 5;*)
		bT_Re_PriCirc_Active : BOOL; (*PARA [13158]: return water temperature primary circuit measurement active*) (*OldName: new PV	; Cycle: 5;*)
		bT_Su_SecCirc_Active : BOOL; (*PARA [13161]: supply water temperature secondary circuit measurement active*) (*OldName: new PV	; Cycle: 5;*)
		bT_Re_SecCirc_Active : BOOL; (*PARA [13164]: return water temperature secondary circuit measurement active*) (*OldName: new PV	; Cycle: 5;*)
		bPos_HW_ReValve : BOOL; (*PARA [13146]: measuring active position control valve heat water return temperature*) (*OldName:newPv; Cycle:5;*)
		bPos_HW_EC_ReValve : BOOL; (*PARA [13147]: measuring active position control valve heat water return temperature after cooler*) (*OldName:newPv; Cycle:5;*)
		bPos_ChCValve : BOOL; (*PARA [13148]: measuring active position control valve charge cooler circuit temperature*) (*OldName:newPv; Cycle:5;*)
		bP_Heat_Active : BOOL; (*PARA [13167]: measuring active heating power engine heat water circuit*) (*OldName:newPv; Cycle:5;*)
		bCnt_P_Heat : BOOL; (*PARA [13170]: counter active heating power engine heat water circuit*) (*OldName:newPv; Cycle:5;*)
		rImpVal_Cnt_P_Heat : REAL; (*PARA [13171]: impulse value counter heating power engine heat water circuit*) (*OldName:newPv; Cycle:5;*)
		bHWF_Active : BOOL; (*PARA [13183]: Kesselhausventilator active*) (*OldName:newPv; Cycle:5;*)
		bCHC_Heating_active : BOOL; (*PARA [13184]: Ladek�hler Vorw�rmung active*) (*OldName:newPv; Cycle:5;*)
		bT_ECW_bChC_HT_Active : BOOL; (*PARA [13395]: temperature engine cooling water before charge cooler high temp.circuit active M.06-TI-014*) (*OldName:newPv; Cycle:5;*)
		bT_ECW_bOilC_Active : BOOL; (*PARA [13396]: temperature engine cooling water before oil cooler active M.06-TI-020*) (*OldName:newPv; Cycle:5;*)
		bT_ECW_bECWC_Active : BOOL; (*PARA [13397]: temperature engine cooling water before engine cooling water cooler active M.06-TI-030*) (*OldName:newPv; Cycle:5;*)
		bBOP_HeatCirc_Act : BOOL; (*PARA [13832]: -Visu: Plant display heat circuit active*) (*OldName:newPv; Cycle:5;*)
		bBOP_EmCoolCirc_Act : BOOL; (*PARA [13833]: -Visu: Plant display emergency cooler circuit active*) (*OldName:newPv; Cycle:5;*)
		bBOP_ChCoolCirc_Act : BOOL; (*PARA [13834]: -Visu: Plant display charge cooling circuit active*) (*OldName:newPv; Cycle:5;*)
		rT_ECW_PwrRamp_LimLo : REAL; (*Para engine cooling water temperature limit low - power limitation for warm up operation [°C]*) (*OldName:newPV; Cycle:5;*)
		iChC2_NumDemAux : INT; (*PARA [14255]: number charge cooler 2 stages with demand auxiliaries*) (*OldName:newPV; Cycle:5;*)
		iChC2_NumStages : INT; (*PARA [14254]: charge cooler 2 number stages*) (*OldName:newPV; Cycle:5;*)
		iChC2_OpMode : INT; (*PARA [14253]: charge cooler 2 operating mode*) (*OldName:newPV; Cycle:5;*)
		iChC2_CtrNum : INT; (*PARA [14256]: charge cooler 2 controller number*) (*OldName:newPV; Cycle:5;*)
		rChC2_ValPosLimHi_On : REAL; (*PARA [14257]: position valve charge cooler 2 ON limit high [%]*) (*OldName:newPV; Cycle:5;*)
		rChC2_ValPosHyHi_On : REAL; (*PARA [14258]: position valve charge cooler 2 ON limit high hysteresis [%]*) (*OldName:newPV; Cycle:5;*)
		rChC2_ValPosLimStageUp : REAL; (*PARA [14259]: position charge cooler 2 valve limit stage up [%]*) (*OldName:newPV; Cycle:5;*)
		rChC2_ValPosLimStageDown : REAL; (*PARA [14260]: position charge cooler 2 valve limit stage down [%]*) (*OldName:newPV; Cycle:5;*)
		tiChC2_DelayOff : TIME; (*PARA [14261]: charge cooler 2 delay OFF*) (*OldName:newPV; Cycle:5;*)
		tiChC2_DelayStageUp : TIME; (*PARA [14262]: charge cooler 2 delay switch stage up *) (*OldName:newPV; Cycle:5;*)
		tiChC2_DelayStageDown : TIME; (*PARA [14263]: charge cooler 2 delay switch stage down*) (*OldName:newPV; Cycle:5;*)
		rT_Ch_T1HP_LimHi1 : REAL; (*PARA [14264]: charge temperature before high-pressure turbocharger high limit 1 [°C]*) (*OldName:newPV; Cycle:5;*)
		rT_Ch_T1HP_LimHi2 : REAL; (*PARA [14267]: charge temperature before high-pressure turbocharger high limit 2 [°C]*) (*OldName:newPV; Cycle:5;*)
		rT_Ch_T1HP_HyHi1 : REAL; (*PARA [14265]: charge temperature before high-pressure turbocharger high hysteresis limit 1 [°C]*) (*OldName:newPV; Cycle:5;*)
		rT_Ch_T1HP_HyHi2 : REAL; (*PARA [14266]: charge temperature before high-pressure turbocharger high hysteresis limit 2 [°C]*) (*OldName:newPV; Cycle:5;*)
		tCtr_ChC_T1HP : _tGeACtrPara; (*Para controller charge temperature before high-pressure turbo charger cooler*) (*OldName:newPV; Cycle:5;*)
		bCtr_ChC_T1HP : BOOL; (*PARA [14244]: visibility charge temperature before high-pressure turbo charger controller*) (*OldName:newPV; Cycle:5;*)
		bAuxChC2_Visible : BOOL; (*PARA [14251]: visibility parameters of charge cooler control*) (*OldName:newPv; Cycle:5;*)
		bChC2_StX_Visible : BOOL; (*PARA [14252]: charge cooler stage0-x visible*) (*OldName:bMixCoolRadStageX; Cycle:5;*)
		bPos_ChC2_Valve : BOOL; (*PARA [14268]: measuring active position control valve 2nd LT charge cooler circuit (T1-HP)*) (*OldName:newPv; Cycle:5;*)
		bT_ChC2_Su_LT_Active : BOOL; (*PARA [14271]: measuring supply water temperature 2nd LT charge cooler circuit (T1-HP) active (P.07-TI-004)*) (*OldName:newPv; Cycle:5;*)
		bT_ChC2_Re_LT_Active : BOOL; (*PARA [14272]: measuring return water temperature 2nd LT charge cooler circuit (T1-HP) active (P.07-TI-006)*) (*OldName:newPv; Cycle:5;*)
		rT_ChC2_Re_LT_LimHi : REAL; (*PARA [14273]: return water temperature 2nd LT charge cooler circuit (T1-HP) maximum*) (*OldName:newPv; Cycle:5;*)
		rT_ChC2_Re_LT_HyHi : REAL; (*PARA [14274]: return water temperature 2nd LT charge cooler circuit (T1-HP) hysteresis*) (*OldName:newPv; Cycle:5;*)
		bChC2_Heating_Active : BOOL; (*PARA [14276]: Ladek�hler 2 Vorw�rmung active*) (*OldName:newPv; Cycle:5;*)
		bEC_Pump_Visible : BOOL; (*PARA [14275]: emergency cooler pump visible*)
		bRedCCWP_Active : BOOL; (*PARA [14347]: Activate redundant pump control for charge cooler water pump *)
		bRedCC2WP_Active : BOOL; (*PARA [14346]: Activate redundant pump control for charge cooler 2 water pump *)
		bRedEmCWP_Active : BOOL; (*PARA [14348]: Activate redundant pump control for emergency cooler water pump *)
		rPr_ECW_LimLo_EngOp : REAL; (*PARA [15066]:Engine cooling water pressure minimum at engine operation*)
		bT_HW_Su_Unit_Active : BOOL; (*PARA [15126]: Heating water supply temperature unit measuring active*) (*SAFETY PLC: newPv; Cycle:5;*) (*V04.25.00.00*)
		rT_HW_Su_Unit_LimHi : REAL; (*PARA [15127]: Heating water supply temperature unit maximum*) (*SAFETY PLC: newPv; Cycle:5;*) (*V04.25.00.00*)
	END_STRUCT;
END_TYPE
```

### module_HC.var - Package variables
```iecst
VAR
	xOpMode : OpMode; (*engine operation mode*)
	xEngType : EngType; (*engine type*)
	xCtr_HWSu : GeACtr; (*heat water supply temperature*)
	xCtr_HWRe : GeACtr; (*heat water return temperature*)
	xCtr_EC : GeACtr; (*emergency cooler*)
	xCtr_ChCV : GeACtr; (*charge cooler ventilation*)
	xCtr_ChCHP : GeACtr; (*charge cooler high pressure*)
	xCtr_ChC : GeACtr; (*charge cooler*)
	xCtr_CDSu : GeACtr; (*condensor circuit supply temperature*)
	VIS2MM : VIS2MM_Struct;
	tCtr_HWSu_Out : _tGeACtrOut; (*heat water supply temperature*)
	tCtr_HWSu_In : _tGeACtrIn; (*heat water supply temperature*)
	tCtr_HWRe_Out : _tGeACtrOut; (*heat water return temperature*)
	tCtr_HWRe_In : _tGeACtrIn; (*heat water return temperature*)
	tCtr_EC_Out : _tGeACtrOut; (*emergency cooler*)
	tCtr_EC_In : _tGeACtrIn; (*emergency cooler*)
	tCtr_ChC_Out : _tGeACtrOut; (*charge cooler*)
	tCtr_ChC_In : _tGeACtrIn; (*charge cooler*)
	tCtr_ChCV_Out : _tGeACtrOut; (*charge cooler ventilation*)
	tCtr_ChCV_In : _tGeACtrIn; (*charge cooler ventilation*)
	tCtr_ChCHP_Out : _tGeACtrOut; (*charge cooler high pressure*)
	tCtr_ChCHP_In : _tGeACtrIn; (*charge cooler high pressure*)
	tCtr_CDSu_Out : _tGeACtrOut; (*condensor circuit supply temperature*)
	tCtr_CDSu_In : _tGeACtrIn; (*condensor circuit supply temperature*)
	pm : PARA_HC_Struct;
	ParaFactoryDefault : PARA_HC_Struct;
	Para : PARA_HC_Struct;
	OUT_HC : OUT_HC_Struct;
	M_KV16 : BOOL; (* Kühler Stufe 16 *)
	M_KV15 : BOOL; (* Kühler Stufe 15 *)
	M_KV14 : BOOL; (* Kühler Stufe 14 *)
	M_KV13 : BOOL; (* Kühler Stufe 13 *)
	M_KV12 : BOOL; (* Kühler Stufe 12 *)
	M_KV11 : BOOL; (* Kühler Stufe 11 *)
	M_KV10 : BOOL; (* Kühler Stufe 10 *)
	M_KV9 : BOOL; (* Kühler Stufe 9 *)
	M_KV8 : BOOL; (* Kühler Stufe 8 *)
	M_KV7 : BOOL; (* Kühler Stufe 7 *)
	M_KV6 : BOOL; (* Kühler Stufe 6 *)
	M_KV5 : BOOL; (* Kühler Stufe 5 *)
	M_KV4 : BOOL; (* Kühler Stufe 4 *)
	M_KV3 : BOOL; (* Kühler Stufe 3 *)
	M_KV2 : BOOL; (* Kühler Stufe 2 *)
	M_KV1 : BOOL; (* Kühler Stufe 1 *)
	M_GKV16 : BOOL; (* Gemischkühler Stufe 16 *)
	M_GKV15 : BOOL; (* Gemischkühler Stufe 15 *)
	M_GKV14 : BOOL; (* Gemischkühler Stufe 14 *)
	M_GKV13 : BOOL; (* Gemischkühler Stufe 13 *)
	M_GKV12 : BOOL; (* Gemischkühler Stufe 12 *)
	M_GKV11 : BOOL; (* Gemischkühler Stufe 11 *)
	M_GKV10 : BOOL; (* Gemischkühler Stufe 10 *)
	M_GKV9 : BOOL; (* Gemischkühler Stufe 9 *)
	M_GKV8 : BOOL; (* Gemischkühler Stufe 8 *)
	M_GKV7 : BOOL; (* Gemischkühler Stufe 7 *)
	M_GKV6 : BOOL; (* Gemischkühler Stufe 6 *)
	M_GKV5 : BOOL; (* Gemischkühler Stufe 5 *)
	M_GKV4 : BOOL; (* Gemischkühler Stufe 4 *)
	M_GKV3 : BOOL; (* Gemischkühler Stufe 3 *)
	M_GKV2 : BOOL; (* Gemischkühler Stufe 2 *)
	M_GKV1 : BOOL; (* Gemischkühler Stufe 1 *)
	MM2VIS : MM2VIS_Struct;
	K_vent : BOOL; (* Stufen abhängig von Ventil *)
	K_temp : BOOL; (* Stufen abhängig von Temperatur *)
	K_ST_16 : BOOL; (* Kühlstufe 16 aktiv *)
	K_ST_15 : BOOL; (* Kühlstufe 15 aktiv *)
	K_ST_14 : BOOL; (* Kühlstufe 14 aktiv *)
	K_ST_13 : BOOL; (* Kühlstufe 13 aktiv *)
	K_ST_12 : BOOL; (* Kühlstufe 12 aktiv *)
	K_ST_11 : BOOL; (* Kühlstufe 11 aktiv *)
	K_ST_10 : BOOL; (* Kühlstufe 10 aktiv *)
	K_ST_9 : BOOL; (* Kühlstufe 9 aktiv *)
	K_ST_8 : BOOL; (* Kühlstufe 8 aktiv *)
	K_ST_7 : BOOL; (* Kühlstufe 7 aktiv *)
	K_ST_6 : BOOL; (* Kühlstufe 6 aktiv *)
	K_ST_5 : BOOL; (* Kühlstufe 5 aktiv *)
	K_ST_4 : BOOL; (* Kühlstufe 4 aktiv *)
	K_ST_3 : BOOL; (* Kühlstufe 3 aktiv *)
	K_ST_2 : BOOL; (* Kühlstufe 2 aktiv *)
	K_ST_1 : BOOL := 1; (* Kühlstufe 1 aktiv *)
	K_ST16 : BOOL; (* Kühler Stufe 16 *)
	K_ST15 : BOOL; (* Kühler Stufe 15 *)
	K_ST14 : BOOL; (* Kühler Stufe 14 *)
	K_ST13 : BOOL; (* Kühler Stufe 13 *)
	K_ST12 : BOOL; (* Kühler Stufe 12 *)
	K_ST11 : BOOL; (* Kühler Stufe 11 *)
	K_ST10 : BOOL; (* Kühler Stufe 10 *)
	K_ST9 : BOOL; (* Kühler Stufe 9 *)
	K_ST8 : BOOL; (* Kühler Stufe 8 *)
	K_ST7 : BOOL; (* Kühler Stufe 7 *)
	K_ST6 : BOOL; (* Kühler Stufe 6 *)
	K_ST5 : BOOL; (* Kühler Stufe 5 *)
	K_ST4 : BOOL; (* Kühler Stufe 4 *)
	K_ST3 : BOOL; (* Kühler Stufe 3 *)
	K_ST2 : BOOL; (*emergency cooler stage 2*)
	K_ST1 : BOOL; (*emergency cooler stage 1*)
	K_PLUS : BOOL; (* Kühlerstufe PLUS *)
	K_MINUS : BOOL; (* Kühlerstufe PLUS *)
	K_EIN : BOOL; (* Kühler EIN *)
	K_anfhbt : BOOL; (* Freigabe Kühler mit ANFHBT *)
	Kombi_K : BOOL := 0; (* Kombikühler *)
	iSumEC_Stages : INT; (*summary emergency cooler stages*)
	iSumChC_Stages : INT; (*summary charge cooler stages*)
	IN_HC : IN_HC_Struct;
	GK_vent : BOOL; (* Stufen abhängig von Ventil *)
	GK_var : USINT; (* charge cooler variation *)
	GK_temp : BOOL; (* Stufen abhängig von Temperatur *)
	GK_ST_16 : BOOL; (* Gemischkühlstufe 16 aktiv *)
	GK_ST_15 : BOOL; (* Gemischkühlstufe 15 aktiv *)
	GK_ST_14 : BOOL; (* Gemischkühlstufe 14 aktiv *)
	GK_ST_13 : BOOL; (* Gemischkühlstufe 13 aktiv *)
	GK_ST_12 : BOOL; (* Gemischkühlstufe 12 aktiv *)
	GK_ST_11 : BOOL; (* Gemischkühlstufe 11 aktiv *)
	GK_ST_10 : BOOL; (* Gemischkühlstufe 10 aktiv *)
	GK_ST_9 : BOOL; (* Gemischkühlstufe 9 aktiv *)
	GK_ST_8 : BOOL; (* Gemischkühlstufe 8 aktiv *)
	GK_ST_7 : BOOL; (* Gemischkühlstufe 7 aktiv *)
	GK_ST_6 : BOOL; (* Gemischkühlstufe 6 aktiv *)
	GK_ST_5 : BOOL; (* Gemischkühlstufe 5 aktiv *)
	GK_ST_4 : BOOL; (* Gemischkühlstufe 4 aktiv *)
	GK_ST_3 : BOOL; (* Gemischkühlstufe 3 aktiv *)
	GK_ST_2 : BOOL; (* Gemischkühlstufe 2 aktiv *)
	GK_ST_1 : BOOL := 1; (* Gemischkühlstufe 1 aktiv *)
	GK_ST16 : BOOL; (* Gemischkühler Stufe 16 *)
	GK_ST15 : BOOL; (* Gemischkühler Stufe 15 *)
	GK_ST14 : BOOL; (* Gemischkühler Stufe 14 *)
	GK_ST13 : BOOL; (* Gemischkühler Stufe 13 *)
	GK_ST12 : BOOL; (* Gemischkühler Stufe 12 *)
	GK_ST11 : BOOL; (* Gemischkühler Stufe 11 *)
	GK_ST10 : BOOL; (* Gemischkühler Stufe 10 *)
	GK_ST9 : BOOL; (* Gemischkühler Stufe 9 *)
	GK_ST8 : BOOL; (* Gemischkühler Stufe 8 *)
	GK_ST7 : BOOL; (* Gemischkühler Stufe 7 *)
	GK_ST6 : BOOL; (* Gemischkühler Stufe 6 *)
	GK_ST5 : BOOL; (* Gemischkühler Stufe 5 *)
	GK_ST4 : BOOL; (* Gemischkühler Stufe 4 *)
	GK_ST3 : BOOL; (* Gemischkühler Stufe 3 *)
	GK_ST2 : BOOL; (* Gemischkühler Stufe 2 *)
	GK_ST1 : BOOL; (* Gemischkühler Stufe 1 *)
	GK_PLUS : BOOL; (* GK-Stufe PLUS *)
	GK_MINUS : BOOL; (* GK-Stufe MINUS *)
	GK_EIN : BOOL; (* Gemischkühler EIN *)
	GK_anz : USINT; (* charge cooler stages *)
	GK_anfhbt : BOOL; (* Freigabe GK mit ANFHBT *)
	bT_HW_Su_HiHi : BOOL; (*temperature heat water supply high high*)
	bT_HW_Su_Hi : BOOL; (*temperature heat water supply high*)
	bT_HW_Re_HiHi : BOOL; (*temperature heat water return high high*)
	bT_HW_Re_Hi : BOOL; (*temperature heat water return high*)
	bT_HW_ReBeEng_HiHi : BOOL; (*temperature heat water return before engine high high*)
	bT_HW_ReBeEng_Hi : BOOL; (*temperature heat water return before engine high*)
	bT_HW_ReAfEC_HiHi : BOOL; (*temperature heat water return after emergency cooler high high*)
	bT_HW_ReAfEC_Hi : BOOL; (*temperature heat water return after emergency cooler high*)
	bT_HW_HC_Re_Hi : BOOL; (*heat circuit tempreature high*)
	bT_Su_PriCirc_Hi : BOOL; (*supply water temperature high primary circuit*)
	bT_Re_PriCirc_Hi : BOOL; (*return water temperature high primary circuit*)
	bT_Su_SecCirc_Hi : BOOL; (*supply water temperature high secondary circuit*)
	bT_Re_SecCirc_Hi : BOOL; (*return water temperature high secondary circuit*)
	bT_EO_Hi2 : BOOL; (* temperature engine oil high *)
	bT_EO_Hi1 : BOOL; (* temperature engine oil high *)
	bT_ECW_HiHi : BOOL; (*temperature engine cooling water high high*)
	bT_ECW_HiHiPrio2 : BOOL; (*temperature engine cooling water high Prio2*)
	bT_ECW_Hi2 : BOOL; (*temperature engine cooling water limit high*)
	bT_ECW_Hi1 : BOOL; (*temperature engine cooling water limit high*)
	bT_Ch_Hi2 : BOOL; (*charge temperature limit high 2*)
	bT_Ch_Hi1 : BOOL; (*charge temperature limit high 1*)
	bT_CD_Su_Hi : BOOL; (*condensor circuit supply temperature high*)
	bT_CD_Re_Hi : BOOL; (*condensor circuit return temperature high*)
	bT_AirOutdoor_Hi4 : BOOL; (* temperature air outdoor limit high *)
	bT_AirOutdoor_Hi3 : BOOL; (* temperature air outdoor limit high *)
	bT_AirOutdoor_Hi2 : BOOL; (* temperature air outdoor limit high *)
	bT_AirOutdoor_Hi1 : BOOL; (* temperature air outdoor limit high *)
	bPr_ECW_LoLo : BOOL; (*pressure engine cooling water low low*)
	bPr_ECW_LimOp : BOOL; (*pressure engine cooling water low during engine operation*)
	bPr_ECW_LoLoPrio2 : BOOL; (*pressure engine cooling water low Prio2*)
	bPr_ECW_Lo : BOOL; (*pressure engine cooling water low*)
	bPr_ECW_HiHi : BOOL; (*pressure engine cooling water high high*)
	bPr_ECW_HiHiPrio2 : BOOL; (*temperature engine cooling water high high Prio 2*)
	bPr_ECW_Hi : BOOL; (*pressure engine cooling water high*)
	bOMSS_Test : BOOL; (*engine operation mode selection*)
	bOMSS_Stop : BOOL; (*engine operation mode selection*)
	bOMSS_Scav : BOOL; (*engine operation mode selection*)
	bOMSS_MAT : BOOL; (*engine operation mode selection*)
	bOMSS_Man : BOOL; (*engine operation mode selection*)
	bOMSS_Aut : BOOL; (*engine operation mode selection*)
	bN_EngStart : BOOL; (*engine start speed*)
	bNoInitDetected : BOOL := FALSE; (*allways true, except 1cycle on init up*)
	bGnlWarning : BOOL; (*general warning*)
	bGnlTrip3 : BOOL; (*general trip 3*)
	bGnlTrip2 : BOOL; (*general trip 2*)
	bGnlTrip1 : BOOL; (*general trip 1*)
	bGnlTrip : BOOL; (*general trip*)
	bFail_BHV : BOOL; (*condensor circuit return temperature high*)
	bEC_Up : BOOL; (*emergency cooler stage up*)
	bEC_Down : BOOL; (*emergency cooler stage down*)
	bECW_DemBpV : BOOL; (*demand engine cooling water bypass valve*)
	bECW_DemBpP : BOOL; (*demand engine cooling water bypass pump*)
	bChC_Up : BOOL; (*charge cooler stage up*)
	bChC_Down : BOOL; (*charge cooler stage down*)
	Anz_GK_anfhbt : USINT; (* Anzahl Stufen GK mit ANFHBT *)
	Anz_anfhbt : USINT; (* Anzahl Stufen Anf. Hilfsbetriebe *)
	K_ST1_ManAuxCtr : BOOL;
	K_ST2_ManAuxCtr : BOOL;
	K_ST3_ManAuxCtr : BOOL;
	K_ST4_ManAuxCtr : BOOL;
	K_ST5_ManAuxCtr : BOOL;
	K_ST6_ManAuxCtr : BOOL;
	K_ST7_ManAuxCtr : BOOL;
	K_ST8_ManAuxCtr : BOOL;
	K_ST9_ManAuxCtr : BOOL;
	K_ST10_ManAuxCtr : BOOL;
	K_ST11_ManAuxCtr : BOOL;
	K_ST12_ManAuxCtr : BOOL;
	K_ST13_ManAuxCtr : BOOL;
	K_ST14_ManAuxCtr : BOOL;
	K_ST15_ManAuxCtr : BOOL;
	K_ST16_ManAuxCtr : BOOL;
	GK_ST1_ManAuxCtr : BOOL;
	GK_ST2_ManAuxCtr : BOOL;
	GK_ST3_ManAuxCtr : BOOL;
	GK_ST4_ManAuxCtr : BOOL;
	GK_ST5_ManAuxCtr : BOOL;
	GK_ST6_ManAuxCtr : BOOL;
	GK_ST7_ManAuxCtr : BOOL;
	GK_ST8_ManAuxCtr : BOOL;
	GK_ST9_ManAuxCtr : BOOL;
	GK_ST10_ManAuxCtr : BOOL;
	GK_ST11_ManAuxCtr : BOOL;
	GK_ST12_ManAuxCtr : BOOL;
	GK_ST13_ManAuxCtr : BOOL;
	GK_ST14_ManAuxCtr : BOOL;
	GK_ST15_ManAuxCtr : BOOL;
	GK_ST16_ManAuxCtr : BOOL;
	bPr_ECW_PcheckFail : BOOL; (*plausibility check measuring signal Pr_ECW*)
	GK2_var : USINT; (* charge cooler 2 variant*)
	GK2_anz : USINT; (* charge cooler 2 stages *)
	Anz_GK2_anfhbt : USINT; (* Anzahl Stufen GK2 mit ANFHBT *)
	bChC2_Up : BOOL; (*charge cooler 2 stage up*)
	bChC2_Down : BOOL; (*charge cooler 2 stage down*)
	bT_Ch2_Hi2 : BOOL; (*charge temperature 2 limit high 2*)
	bT_Ch2_Hi1 : BOOL; (*charge temperature 2 limit high 1*)
	GK2_vent : BOOL; (* Stufen abhängig von Ventil - charge cooler 2*)
	GK2_temp : BOOL; (* Stufen abhängig von Temperatur - charge cooler 2 *)
	GK2_anfhbt : BOOL; (* Freigabe GK2 mit ANFHBT *)
	GK2_ST_16 : BOOL; (* Gemischkühler 2 Stufe 16 aktiv *)
	GK2_ST_15 : BOOL; (* Gemischkühler 2 Stufe 15 aktiv *)
	GK2_ST_14 : BOOL; (* Gemischkühler 2 Stufe 14 aktiv *)
	GK2_ST_13 : BOOL; (* Gemischkühler 2 Stufe 13 aktiv *)
	GK2_ST_12 : BOOL; (* Gemischkühler 2 Stufe 12 aktiv *)
	GK2_ST_11 : BOOL; (* Gemischkühler 2 Stufe 11 aktiv *)
	GK2_ST_10 : BOOL; (* Gemischkühler 2 Stufe 10 aktiv *)
	GK2_ST_9 : BOOL; (* Gemischkühler 2 Stufe 9 aktiv *)
	GK2_ST_8 : BOOL; (* Gemischkühler 2 Stufe 8 aktiv *)
	GK2_ST_7 : BOOL; (* Gemischkühler 2 Stufe 7 aktiv *)
	GK2_ST_6 : BOOL; (* Gemischkühler 2 Stufe 6 aktiv *)
	GK2_ST_5 : BOOL; (* Gemischkühler 2 Stufe 5 aktiv *)
	GK2_ST_4 : BOOL; (* Gemischkühler 2 Stufe 4 aktiv *)
	GK2_ST_3 : BOOL; (* Gemischkühler 2 Stufe 3 aktiv *)
	GK2_ST_2 : BOOL; (* Gemischkühler 2 Stufe 2 aktiv *)
	GK2_ST_1 : BOOL := 1; (* Gemischkühler 2 Stufe 1 aktiv *)
	GK2_EIN : BOOL; (* Gemischkühler 2 EIN *)
	GK2_PLUS : BOOL; (* GK2-Stufe PLUS *)
	GK2_MINUS : BOOL; (* GK2-Stufe MINUS *)
	M_GK2V16 : BOOL; (* Gemischkühler 2 Stufe 16 *)
	M_GK2V15 : BOOL; (* Gemischkühler 2 Stufe 15 *)
	M_GK2V14 : BOOL; (* Gemischkühler 2 Stufe 14 *)
	M_GK2V13 : BOOL; (* Gemischkühler 2 Stufe 13 *)
	M_GK2V12 : BOOL; (* Gemischkühler 2 Stufe 12 *)
	M_GK2V11 : BOOL; (* Gemischkühler 2 Stufe 11 *)
	M_GK2V10 : BOOL; (* Gemischkühler 2 Stufe 10 *)
	M_GK2V9 : BOOL; (* Gemischkühler 2 Stufe 9 *)
	M_GK2V8 : BOOL; (* Gemischkühler 2 Stufe 8 *)
	M_GK2V7 : BOOL; (* Gemischkühler 2 Stufe 7 *)
	M_GK2V6 : BOOL; (* Gemischkühler 2 Stufe 6 *)
	M_GK2V5 : BOOL; (* Gemischkühler 2 Stufe 5 *)
	M_GK2V4 : BOOL; (* Gemischkühler 2 Stufe 4 *)
	M_GK2V3 : BOOL; (* Gemischkühler 2 Stufe 3 *)
	M_GK2V2 : BOOL; (* Gemischkühler 2 Stufe 2 *)
	M_GK2V1 : BOOL; (* Gemischkühler 2 Stufe 1 *)
	GK2_ST16 : BOOL; (* Gemischkühler 2 Stufe 16 *)
	GK2_ST15 : BOOL; (* Gemischkühler 2 Stufe 15 *)
	GK2_ST14 : BOOL; (* Gemischkühler 2 Stufe 14 *)
	GK2_ST13 : BOOL; (* Gemischkühler 2 Stufe 13 *)
	GK2_ST12 : BOOL; (* Gemischkühler 2 Stufe 12 *)
	GK2_ST11 : BOOL; (* Gemischkühler 2 Stufe 11 *)
	GK2_ST10 : BOOL; (* Gemischkühler 2 Stufe 10 *)
	GK2_ST9 : BOOL; (* Gemischkühler 2 Stufe 9 *)
	GK2_ST8 : BOOL; (* Gemischkühler 2 Stufe 8 *)
	GK2_ST7 : BOOL; (* Gemischkühler 2 Stufe 7 *)
	GK2_ST6 : BOOL; (* Gemischkühler 2 Stufe 6 *)
	GK2_ST5 : BOOL; (* Gemischkühler 2 Stufe 5 *)
	GK2_ST4 : BOOL; (* Gemischkühler 2 Stufe 4 *)
	GK2_ST3 : BOOL; (* Gemischkühler 2 Stufe 3 *)
	GK2_ST2 : BOOL; (* Gemischkühler 2 Stufe 2 *)
	GK2_ST1 : BOOL; (* Gemischkühler 2 Stufe 1 *)
	tCtr_ChC_T1HP_Out : _tGeACtrOut; (*charge cooler 2*)
	tCtr_ChC_T1HP_In : _tGeACtrIn; (*charge cooler 2*)
	xCtr_ChC_T1HP : GeACtr; (*charge cooler 2*)
	GK2_ST1_ManAuxCtr : BOOL;
	GK2_ST2_ManAuxCtr : BOOL;
	GK2_ST3_ManAuxCtr : BOOL;
	GK2_ST4_ManAuxCtr : BOOL;
	GK2_ST5_ManAuxCtr : BOOL;
	GK2_ST6_ManAuxCtr : BOOL;
	GK2_ST7_ManAuxCtr : BOOL;
	GK2_ST8_ManAuxCtr : BOOL;
	GK2_ST9_ManAuxCtr : BOOL;
	GK2_ST10_ManAuxCtr : BOOL;
	GK2_ST11_ManAuxCtr : BOOL;
	GK2_ST12_ManAuxCtr : BOOL;
	GK2_ST13_ManAuxCtr : BOOL;
	GK2_ST14_ManAuxCtr : BOOL;
	GK2_ST15_ManAuxCtr : BOOL;
	GK2_ST16_ManAuxCtr : BOOL;
	iSumChC2_Stages : INT; (*summary charge cooler 2 stages*)
	bECW_ShutOffVal_Dem_Exist : BOOL; (*demand 2-way shut off valve engine jacket water circuit exist*)
	bValHeater_Dem_Exist : BOOL; (*demand 3-way valve heater exist*)
	bFanRingHeater_Dem_Exist : BOOL; (*demand fan ring heater exist*)
END_VAR
```

### Program Logical/HeatingCooling/default_HC (IEC, version 4.11.0) - values

#### default_HCCyclic.st
```iecst
(*******************************************************************************
default		value set

This code is confidential and proprietary to the INNIO Company.
It may not be used in any form, or reproduced in any manner,
without the express written permission of the INNIO Company.
Copyright, INNIO Company, 2019

Customized modifications: -
------------------------

History:
-------
V3.99.0	24.04.2012	lettenb.	new
V4.00.0 14.04.2015				tChC_FanRdy added
V4.03.0 30.09.2015	plattner	tHWF_Fail, tAuxV_Aux_Ok, tAuxV_ModIf_ok, tCDP_Op added
V4.07.0	09.08.2018	Schmid		2nd low temperature charge cooling circuit added
V4.11.0	28.01.2022	Schmid		tECWP_Op added

Instructions for use:
--------------------
Outstandings:
------------
*******************************************************************************)
PROGRAM _CYCLIC

	(* default TRUE setting for not existing Di's *)
	IN_HC.tFlow_HW_Lo.Di			:=	IN_HC.tFlow_HW_Lo.Di			OR	NOT IN_HC.tFlow_HW_Lo.GoodQual;
	IN_HC.tPr_ChC_Lo.Di				:=	IN_HC.tPr_ChC_Lo.Di				OR	NOT IN_HC.tPr_ChC_Lo.GoodQual;
	IN_HC.tPr_ChC2_Lo.Di			:=	IN_HC.tPr_ChC2_Lo.Di			OR	NOT IN_HC.tPr_ChC2_Lo.GoodQual;
	IN_HC.tEC_Failure.Di			:=	IN_HC.tEC_Failure.Di			OR	NOT IN_HC.tEC_Failure.GoodQual;
	IN_HC.tChC_Failure.Di			:=	IN_HC.tChC_Failure.Di			OR	NOT IN_HC.tChC_Failure.GoodQual;
	IN_HC.tChC2_Failure.Di			:=	IN_HC.tChC2_Failure.Di			OR	NOT IN_HC.tChC2_Failure.GoodQual;
	IN_HC.tPr_CCircuit_Lo.Di		:=	IN_HC.tPr_CCircuit_Lo.Di		OR	NOT IN_HC.tPr_CCircuit_Lo.GoodQual;
	IN_HC.tT_ChCW_Hi.Di				:=	IN_HC.tT_ChCW_Hi.Di				OR	NOT IN_HC.tT_ChCW_Hi.GoodQual;
	IN_HC.tT_ChC2W_Hi.Di			:=	IN_HC.tT_ChC2W_Hi.Di			OR	NOT IN_HC.tT_ChC2W_Hi.GoodQual;
	IN_HC.tChC_FanRdy.Di			:=	IN_HC.tChC_FanRdy.Di			OR	NOT IN_HC.tChC_FanRdy.GoodQual;
	IN_HC.tChC2_FanRdy.Di			:=	IN_HC.tChC2_FanRdy.Di			OR	NOT IN_HC.tChC2_FanRdy.GoodQual;
	IN_HC.tAuxV_Aux_ok.Di			:=	IN_HC.tAuxV_Aux_ok.Di			OR	NOT IN_HC.tAuxV_Aux_ok.GoodQual;
	IN_HC.tAuxV_ModIf_ok.Di			:=	IN_HC.tAuxV_ModIf_ok.Di			OR	NOT IN_HC.tAuxV_ModIf_ok.GoodQual;
	IN_HC.tHWF_Fail.Di				:=	IN_HC.tHWF_Fail.Di				OR	NOT IN_HC.tHWF_Fail.GoodQual;
	IN_HC.tCDP_Op.Di				:=	IN_HC.tCDP_Op.Di				OR	NOT IN_HC.tCDP_Op.GoodQual;
	IN_HC.tECWP_Op.Di				:=	IN_HC.tECWP_Op.Di				OR	NOT IN_HC.tECWP_Op.GoodQual;

	//	IN_HC.x.Di		:=	IN_HC.x.Di		OR	NOT IN_HC.x.GoodQual;

END_PROGRAM
```

### Program Logical/HeatingCooling/general_HC (IEC, version 4.14.0) - functions
